LIN {X 0,Y 438.701,Z 233.838,A -85,B 0,C 180,E1 -9266.355,E2 -9266.355} C_VEL
LIN {X 0,Y 435.885,Z 234.19,A -85,B 0,C 180,E1 -9267.602,E2 -9267.602} C_VEL
LIN {X 0,Y 433.569,Z 234.475,A -85,B 0,C 180,E1 -9268.609,E2 -9268.609} C_VEL
LIN {X 0,Y 432.642,Z 234.593,A -85,B 0,C 180,E1 -9269.385,E2 -9269.385} C_VEL
LIN {X 0,Y 432.601,Z 234.596,A -85,B 0,C 180,E1 -9269.648,E2 -9269.648} C_VEL
LIN {X 0,Y 432.582,Z 234.598,A -85,B 0,C 180,E1 -9272.794,E2 -9272.794} C_VEL
LIN {X 0,Y 432.228,Z 234.848,A -85,B 0,C 180,E1 -9275.833,E2 -9275.833} C_VEL
LIN {X 0,Y 432.01,Z 242.324,A -85,B 0,C 180,E1 -9279.362,E2 -9279.362} C_VEL
LIN {X 0,Y 432.001,Z 248.987,A -85,B 0,C 180,E1 -9282.548,E2 -9282.548} C_VEL
LIN {X 0,Y 431.835,Z 256.608,A -85,B 0,C 180,E1 -9286.216,E2 -9286.216} C_VEL
LIN {X 0,Y 431.743,Z 262.883,A -85,B 0,C 180,E1 -9289.241,E2 -9289.241} C_VEL
LIN {X 0,Y 431.628,Z 270.665,A -85,B 0,C 180,E1 -9293.003,E2 -9293.003} C_VEL
LIN {X 0,Y 431.636,Z 272.767,A -85,B 0,C 180,E1 -9294.02,E2 -9294.02} C_VEL
LIN {X 0,Y 433.636,Z 283.694,A -85,B 0,C 180,E1 -9294.477,E2 -9294.477} C_VEL
LIN {X 0,Y 434.113,Z 288.557,A -85,B 0,C 180,E1 -9294.726,E2 -9294.726} C_VEL
LIN {X 0,Y 433.839,Z 297.433,A -85,B 0,C 180,E1 -9295.244,E2 -9295.244} C_VEL
LIN {X 0,Y 433.543,Z 305.193,A -85,B 0,C 180,E1 -9295.814,E2 -9295.814} C_VEL
LIN {X 0,Y 433.148,Z 313.826,A -85,B 0,C 180,E1 -9296.601,E2 -9296.601} C_VEL
LIN {X 0,Y 432.757,Z 322.389,A -85,B 0,C 180,E1 -9297.571,E2 -9297.571} C_VEL
LIN {X 0,Y 432.408,Z 329.809,A -85,B 0,C 180,E1 -9298.637,E2 -9298.637} C_VEL
LIN {X 0,Y 432.074,Z 335.997,A -85,B 0,C 180,E1 -9299.743,E2 -9299.743} C_VEL
LIN {X 0,Y 431.833,Z 341.036,A -85,B 0,C 180,E1 -9300.859,E2 -9300.859} C_VEL
LIN {X 0,Y 431.636,Z 344.371,A -85,B 0,C 180,E1 -9301.763,E2 -9301.763} C_VEL
LIN {X 0,Y 431.505,Z 346.73,A -85,B 0,C 180,E1 -9302.512,E2 -9302.512} C_VEL
LIN {X 0,Y 431.395,Z 349.76,A -85,B 0,C 180,E1 -9303.813,E2 -9303.813} C_VEL
LIN {X 0,Y 431.27,Z 351.381,A -85,B 0,C 180,E1 -9304.776,E2 -9304.776} C_VEL
LIN {X 0,Y 431.202,Z 352.556,A -85,B 0,C 180,E1 -9305.927,E2 -9305.927} C_VEL
LIN {X 0,Y 431.197,Z 352.968,A -85,B 0,C 180,E1 -9307.089,E2 -9307.089} C_VEL
LIN {X 0,Y 431.208,Z 352.366,A -85,B 0,C 180,E1 -9308.526,E2 -9308.526} C_VEL
LIN {X 0,Y 431.279,Z 351.408,A -85,B 0,C 180,E1 -9309.46,E2 -9309.46} C_VEL
LIN {X 0,Y 431.441,Z 349.345,A -85,B 0,C 180,E1 -9310.661,E2 -9310.661} C_VEL
LIN {X 0,Y 431.614,Z 346.292,A -85,B 0,C 180,E1 -9311.883,E2 -9311.883} C_VEL
LIN {X 0,Y 431.882,Z 342.137,A -85,B 0,C 180,E1 -9313.115,E2 -9313.115} C_VEL
LIN {X 0,Y 432.092,Z 337.011,A -85,B 0,C 180,E1 -9314.302,E2 -9314.302} C_VEL
LIN {X 0,Y 432.515,Z 329.674,A -85,B 0,C 180,E1 -9315.64,E2 -9315.64} C_VEL
LIN {X 0,Y 432.986,Z 321.729,A -85,B 0,C 180,E1 -9316.751,E2 -9316.751} C_VEL
LIN {X 0,Y 433.309,Z 314.409,A -85,B 0,C 180,E1 -9317.583,E2 -9317.583} C_VEL
LIN {X 0,Y 433.726,Z 306.857,A -85,B 0,C 180,E1 -9318.285,E2 -9318.285} C_VEL
LIN {X 0,Y 434.003,Z 298.823,A -85,B 0,C 180,E1 -9318.897,E2 -9318.897} C_VEL
LIN {X 0,Y 434.321,Z 289.976,A -85,B 0,C 180,E1 -9319.428,E2 -9319.428} C_VEL
LIN {X 0,Y 434.102,Z 286.131,A -85,B 0,C 180,E1 -9319.639,E2 -9319.639} C_VEL
LIN {X 0,Y 432.039,Z 274.897,A -85,B 0,C 180,E1 -9320.135,E2 -9320.135} C_VEL
LIN {X 0,Y 431.73,Z 273.307,A -85,B 0,C 180,E1 -9320.214,E2 -9320.214} C_VEL
LIN {X 0,Y 431.807,Z 266.369,A -85,B 0,C 180,E1 -9323.554,E2 -9323.554} C_VEL
LIN {X 0,Y 431.884,Z 260.379,A -85,B 0,C 180,E1 -9326.407,E2 -9326.407} C_VEL
LIN {X 0,Y 431.963,Z 255.691,A -85,B 0,C 180,E1 -9328.625,E2 -9328.625} C_VEL
LIN {X 0,Y 432.054,Z 249.71,A -85,B 0,C 180,E1 -9331.449,E2 -9331.449} C_VEL
LIN {X 0,Y 432.147,Z 241.916,A -85,B 0,C 180,E1 -9334.986,E2 -9334.986} C_VEL
LIN {X 0,Y 432.217,Z 234.655,A -85,B 0,C 180,E1 -9338.289,E2 -9338.289} C_VEL
LIN {X 0,Y 432.386,Z 234.628,A -85,B 0,C 180,E1 -9341.029,E2 -9341.029} C_VEL
LIN {X 0,Y 432.433,Z 234.621,A -85,B 0,C 180,E1 -9343.961,E2 -9343.961} C_VEL
LIN {X 0,Y 432.462,Z 234.619,A -85,B 0,C 180,E1 -9347.803,E2 -9347.803} C_VEL
LIN {X 0,Y 432.486,Z 234.615,A -85,B 0,C 180,E1 -9351.59,E2 -9351.59} C_VEL
LIN {X 0,Y 432.583,Z 234.603,A -85,B 0,C 180,E1 -9354.406,E2 -9354.406} C_VEL
LIN {X 0,Y 432.607,Z 234.599,A -85,B 0,C 180,E1 -9358.138,E2 -9358.138} C_VEL
LIN {X 0,Y 432.735,Z 234.583,A -85,B 0,C 180,E1 -9360,E2 -9360} C_VEL
LIN {X 0,Y 432.594,Z 234.601,A -85,B 0,C 180,E1 -9362.794,E2 -9362.794} C_VEL
LIN {X 0,Y 432.588,Z 234.601,A -85,B 0,C 180,E1 -9365.594,E2 -9365.594} C_VEL
LIN {X 0,Y 432.485,Z 234.614,A -85,B 0,C 180,E1 -9368.41,E2 -9368.41} C_VEL
LIN {X 0,Y 432.462,Z 234.618,A -85,B 0,C 180,E1 -9372.196,E2 -9372.196} C_VEL
LIN {X 0,Y 432.433,Z 234.618,A -85,B 0,C 180,E1 -9376.039,E2 -9376.039} C_VEL
LIN {X 0,Y 432.389,Z 234.626,A -85,B 0,C 180,E1 -9379.485,E2 -9379.485} C_VEL
LIN {X 0,Y 432.319,Z 234.635,A -85,B 0,C 180,E1 -9382.964,E2 -9382.964} C_VEL
LIN {X 0,Y 432.352,Z 234.631,A -85,B 0,C 180,E1 -9386.033,E2 -9386.033} C_VEL
LIN {X 0,Y 432.344,Z 234.629,A -85,B 0,C 180,E1 -9389.187,E2 -9389.187} C_VEL
LIN {X 0,Y 432.324,Z 234.634,A -85,B 0,C 180,E1 -9392.443,E2 -9392.443} C_VEL
LIN {X 0,Y 432.344,Z 234.631,A -85,B 0,C 180,E1 -9395.632,E2 -9395.632} C_VEL
LIN {X 0,Y 432.352,Z 234.63,A -85,B 0,C 180,E1 -9399.343,E2 -9399.343} C_VEL
LIN {X 0,Y 432.335,Z 234.632,A -85,B 0,C 180,E1 -9401.797,E2 -9401.797} C_VEL
LIN {X 0,Y 432.335,Z 234.634,A -85,B 0,C 180,E1 -9404.347,E2 -9404.347} C_VEL
LIN {X 0,Y 432.321,Z 234.636,A -85,B 0,C 180,E1 -9407.016,E2 -9407.016} C_VEL
LIN {X 0,Y 432.379,Z 234.679,A -85,B 0,C 180,E1 -9408.391,E2 -9408.391} C_VEL
LIN {X 0,Y 433.342,Z 240.284,A -85,B 0,C 180,E1 -9411.121,E2 -9411.121} C_VEL
LIN {X 0,Y 434.088,Z 244.688,A -85,B 0,C 180,E1 -9413.199,E2 -9413.199} C_VEL
LIN {X 0,Y 434.184,Z 248.536,A -85,B 0,C 180,E1 -9414.926,E2 -9414.926} C_VEL
LIN {X 0,Y 433.596,Z 256.21,A -85,B 0,C 180,E1 -9418.212,E2 -9418.212} C_VEL
LIN {X 0,Y 432.942,Z 265.131,A -85,B 0,C 180,E1 -9421.916,E2 -9421.916} C_VEL
LIN {X 0,Y 432.55,Z 272.79,A -85,B 0,C 180,E1 -9425.011,E2 -9425.011} C_VEL
LIN {X 0,Y 432.083,Z 281.721,A -85,B 0,C 180,E1 -9428.533,E2 -9428.533} C_VEL
LIN {X 0,Y 431.788,Z 289.361,A -85,B 0,C 180,E1 -9431.495,E2 -9431.495} C_VEL
LIN {X 0,Y 431.664,Z 294.798,A -85,B 0,C 180,E1 -9433.555,E2 -9433.555} C_VEL
LIN {X 0,Y 433.565,Z 308.82,A -85,B 0,C 180,E1 -9434.065,E2 -9434.065} C_VEL
LIN {X 0,Y 434.856,Z 320.587,A -85,B 0,C 180,E1 -9434.654,E2 -9434.654} C_VEL
LIN {X 0,Y 434.294,Z 332.166,A -85,B 0,C 180,E1 -9435.354,E2 -9435.354} C_VEL
LIN {X 0,Y 433.643,Z 344.096,A -85,B 0,C 180,E1 -9436.273,E2 -9436.273} C_VEL
LIN {X 0,Y 433.051,Z 355.074,A -85,B 0,C 180,E1 -9437.344,E2 -9437.344} C_VEL
LIN {X 0,Y 432.508,Z 364.833,A -85,B 0,C 180,E1 -9438.518,E2 -9438.518} C_VEL
LIN {X 0,Y 432.017,Z 372.866,A -85,B 0,C 180,E1 -9439.692,E2 -9439.692} C_VEL
LIN {X 0,Y 431.665,Z 380.764,A -85,B 0,C 180,E1 -9441.102,E2 -9441.102} C_VEL
LIN {X 0,Y 431.463,Z 387.072,A -85,B 0,C 180,E1 -9442.513,E2 -9442.513} C_VEL
LIN {X 0,Y 431.296,Z 392.342,A -85,B 0,C 180,E1 -9444.008,E2 -9444.008} C_VEL
LIN {X 0,Y 431.283,Z 395.91,A -85,B 0,C 180,E1 -9445.327,E2 -9445.327} C_VEL
LIN {X 0,Y 431.238,Z 397.871,A -85,B 0,C 180,E1 -9446.262,E2 -9446.262} C_VEL
LIN {X 0,Y 431.318,Z 399.408,A -85,B 0,C 180,E1 -9447.198,E2 -9447.198} C_VEL
LIN {X 0,Y 431.285,Z 400.463,A -85,B 0,C 180,E1 -9448.132,E2 -9448.132} C_VEL
LIN {X 0,Y 431.292,Z 401.104,A -85,B 0,C 180,E1 -9449.066,E2 -9449.066} C_VEL
LIN {X 0,Y 431.283,Z 401.338,A -85,B 0,C 180,E1 -9450,E2 -9450} C_VEL
LIN {X 0,Y 431.262,Z 401.157,A -85,B 0,C 180,E1 -9450.934,E2 -9450.934} C_VEL
LIN {X 0,Y 431.274,Z 400.52,A -85,B 0,C 180,E1 -9451.868,E2 -9451.868} C_VEL
LIN {X 0,Y 431.318,Z 399.475,A -85,B 0,C 180,E1 -9452.802,E2 -9452.802} C_VEL
LIN {X 0,Y 431.23,Z 398.014,A -85,B 0,C 180,E1 -9453.738,E2 -9453.738} C_VEL
LIN {X 0,Y 431.322,Z 394.966,A -85,B 0,C 180,E1 -9455.142,E2 -9455.142} C_VEL
LIN {X 0,Y 431.376,Z 390.847,A -85,B 0,C 180,E1 -9456.549,E2 -9456.549} C_VEL
LIN {X 0,Y 431.582,Z 384.552,A -85,B 0,C 180,E1 -9458.192,E2 -9458.192} C_VEL
LIN {X 0,Y 431.856,Z 377.702,A -85,B 0,C 180,E1 -9459.602,E2 -9459.602} C_VEL
LIN {X 0,Y 432.322,Z 369.259,A -85,B 0,C 180,E1 -9461.012,E2 -9461.012} C_VEL
LIN {X 0,Y 432.9,Z 360.702,A -85,B 0,C 180,E1 -9462.184,E2 -9462.184} C_VEL
LIN {X 0,Y 433.391,Z 351.217,A -85,B 0,C 180,E1 -9463.267,E2 -9463.267} C_VEL
LIN {X 0,Y 434.171,Z 340.199,A -85,B 0,C 180,E1 -9464.292,E2 -9464.292} C_VEL
LIN {X 0,Y 435.046,Z 327.759,A -85,B 0,C 180,E1 -9465.219,E2 -9465.219} C_VEL
LIN {X 0,Y 435.258,Z 320.109,A -85,B 0,C 180,E1 -9465.692,E2 -9465.692} C_VEL
LIN {X 0,Y 434.242,Z 307.284,A -85,B 0,C 180,E1 -9466.395,E2 -9466.395} C_VEL
LIN {X 0,Y 432.159,Z 294.828,A -85,B 0,C 180,E1 -9466.968,E2 -9466.968} C_VEL
LIN {X 0,Y 431.597,Z 291.722,A -85,B 0,C 180,E1 -9467.105,E2 -9467.105} C_VEL
LIN {X 0,Y 431.878,Z 282.941,A -85,B 0,C 180,E1 -9470.48,E2 -9470.48} C_VEL
LIN {X 0,Y 432.213,Z 275.478,A -85,B 0,C 180,E1 -9473.477,E2 -9473.477} C_VEL
LIN {X 0,Y 432.667,Z 267.899,A -85,B 0,C 180,E1 -9476.697,E2 -9476.697} C_VEL
LIN {X 0,Y 433.186,Z 261.43,A -85,B 0,C 180,E1 -9479.659,E2 -9479.659} C_VEL
LIN {X 0,Y 433.901,Z 255.542,A -85,B 0,C 180,E1 -9482.621,E2 -9482.621} C_VEL
LIN {X 0,Y 434.361,Z 252.169,A -85,B 0,C 180,E1 -9484.493,E2 -9484.493} C_VEL
LIN {X 0,Y 434.538,Z 248.602,A -85,B 0,C 180,E1 -9486.757,E2 -9486.757} C_VEL
LIN {X 0,Y 434.258,Z 245.52,A -85,B 0,C 180,E1 -9489.137,E2 -9489.137} C_VEL
LIN {X 0,Y 433.805,Z 242.819,A -85,B 0,C 180,E1 -9491.82,E2 -9491.82} C_VEL
LIN {X 0,Y 433.477,Z 240.907,A -85,B 0,C 180,E1 -9494.49,E2 -9494.49} C_VEL
LIN {X 0,Y 433.227,Z 239.772,A -85,B 0,C 180,E1 -9497.051,E2 -9497.051} C_VEL
LIN {X 0,Y 433.123,Z 239.257,A -85,B 0,C 180,E1 -9499.698,E2 -9499.698} C_VEL
LIN {X 0,Y 433.098,Z 239.446,A -85,B 0,C 180,E1 -9503.101,E2 -9503.101} C_VEL
LIN {X 0,Y 433.01,Z 240.207,A -85,B 0,C 180,E1 -9505.87,E2 -9505.87} C_VEL
LIN {X 0,Y 432.715,Z 241.447,A -85,B 0,C 180,E1 -9508.686,E2 -9508.686} C_VEL
LIN {X 0,Y 432.439,Z 243.225,A -85,B 0,C 180,E1 -9511.881,E2 -9511.881} C_VEL
LIN {X 0,Y 432.306,Z 244.571,A -85,B 0,C 180,E1 -9513.964,E2 -9513.964} C_VEL
LIN {X 0,Y 432.089,Z 246.753,A -85,B 0,C 180,E1 -9517.023,E2 -9517.023} C_VEL
LIN {X 0,Y 431.942,Z 249.63,A -85,B 0,C 180,E1 -9520.684,E2 -9520.684} C_VEL
LIN {X 0,Y 431.881,Z 252.494,A -85,B 0,C 180,E1 -9524.061,E2 -9524.061} C_VEL
LIN {X 0,Y 435.436,Z 264.773,A -85,B 0,C 180,E1 -9524.753,E2 -9524.753} C_VEL
LIN {X 0,Y 436.678,Z 271.049,A -85,B 0,C 180,E1 -9525.137,E2 -9525.137} C_VEL
LIN {X 0,Y 435.976,Z 283.695,A -85,B 0,C 180,E1 -9525.887,E2 -9525.887} C_VEL
LIN {X 0,Y 435.237,Z 295.639,A -85,B 0,C 180,E1 -9526.816,E2 -9526.816} C_VEL
LIN {X 0,Y 434.487,Z 306.414,A -85,B 0,C 180,E1 -9527.861,E2 -9527.861} C_VEL
LIN {X 0,Y 433.871,Z 316.104,A -85,B 0,C 180,E1 -9529.028,E2 -9529.028} C_VEL
LIN {X 0,Y 433.179,Z 325.539,A -85,B 0,C 180,E1 -9530.427,E2 -9530.427} C_VEL
LIN {X 0,Y 432.616,Z 333.133,A -85,B 0,C 180,E1 -9531.828,E2 -9531.828} C_VEL
LIN {X 0,Y 432.043,Z 340.11,A -85,B 0,C 180,E1 -9533.462,E2 -9533.462} C_VEL
LIN {X 0,Y 431.926,Z 344.73,A -85,B 0,C 180,E1 -9534.866,E2 -9534.866} C_VEL
LIN {X 0,Y 431.807,Z 348.254,A -85,B 0,C 180,E1 -9536.267,E2 -9536.267} C_VEL
LIN {X 0,Y 431.621,Z 350.072,A -85,B 0,C 180,E1 -9537.2,E2 -9537.2} C_VEL
LIN {X 0,Y 431.429,Z 351.421,A -85,B 0,C 180,E1 -9538.133,E2 -9538.133} C_VEL
LIN {X 0,Y 431.292,Z 352.894,A -85,B 0,C 180,E1 -9540,E2 -9540} C_VEL
LIN {X 0,Y 431.316,Z 353.025,A -85,B 0,C 180,E1 -9540.934,E2 -9540.934} C_VEL
LIN {X 0,Y 431.395,Z 352.011,A -85,B 0,C 180,E1 -9542.802,E2 -9542.802} C_VEL
LIN {X 0,Y 431.442,Z 350.912,A -85,B 0,C 180,E1 -9543.736,E2 -9543.736} C_VEL
LIN {X 0,Y 431.389,Z 349.378,A -85,B 0,C 180,E1 -9544.672,E2 -9544.672} C_VEL
LIN {X 0,Y 431.596,Z 346.24,A -85,B 0,C 180,E1 -9546.076,E2 -9546.076} C_VEL
LIN {X 0,Y 431.705,Z 342.027,A -85,B 0,C 180,E1 -9547.483,E2 -9547.483} C_VEL
LIN {X 0,Y 432.065,Z 335.576,A -85,B 0,C 180,E1 -9549.125,E2 -9549.125} C_VEL
LIN {X 0,Y 432.393,Z 328.569,A -85,B 0,C 180,E1 -9550.536,E2 -9550.536} C_VEL
LIN {X 0,Y 432.936,Z 319.801,A -85,B 0,C 180,E1 -9551.945,E2 -9551.945} C_VEL
LIN {X 0,Y 433.438,Z 309.685,A -85,B 0,C 180,E1 -9553.261,E2 -9553.261} C_VEL
LIN {X 0,Y 433.962,Z 299.835,A -85,B 0,C 180,E1 -9554.299,E2 -9554.299} C_VEL
LIN {X 0,Y 434.644,Z 288.818,A -85,B 0,C 180,E1 -9555.234,E2 -9555.234} C_VEL
LIN {X 0,Y 435.221,Z 276.122,A -85,B 0,C 180,E1 -9556.09,E2 -9556.09} C_VEL
LIN {X 0,Y 435.287,Z 267.404,A -85,B 0,C 180,E1 -9556.556,E2 -9556.556} C_VEL
LIN {X 0,Y 432.494,Z 254.275,A -85,B 0,C 180,E1 -9557.189,E2 -9557.189} C_VEL
LIN {X 0,Y 431.416,Z 249.122,A -85,B 0,C 180,E1 -9557.406,E2 -9557.406} C_VEL
LIN {X 0,Y 431.412,Z 246.253,A -85,B 0,C 180,E1 -9560.005,E2 -9560.005} C_VEL
LIN {X 0,Y 431.424,Z 242.986,A -85,B 0,C 180,E1 -9563.015,E2 -9563.015} C_VEL
LIN {X 0,Y 431.602,Z 239.361,A -85,B 0,C 180,E1 -9566.414,E2 -9566.414} C_VEL
LIN {X 0,Y 431.597,Z 236.411,A -85,B 0,C 180,E1 -9569.243,E2 -9569.243} C_VEL
LIN {X 0,Y 431.615,Z 235.278,A -85,B 0,C 180,E1 -9570.344,E2 -9570.344} C_VEL
LIN {X 0,Y 431.687,Z 234.716,A -85,B 0,C 180,E1 -9571.398,E2 -9571.398} C_VEL
LIN {X 0,Y 432.087,Z 234.664,A -85,B 0,C 180,E1 -9574.701,E2 -9574.701} C_VEL
LIN {X 0,Y 432.29,Z 234.637,A -85,B 0,C 180,E1 -9577.191,E2 -9577.191} C_VEL
LIN {X 0,Y 432.336,Z 234.631,A -85,B 0,C 180,E1 -9580.179,E2 -9580.179} C_VEL
LIN {X 0,Y 432.318,Z 234.634,A -85,B 0,C 180,E1 -9583.061,E2 -9583.061} C_VEL
LIN {X 0,Y 432.336,Z 234.631,A -85,B 0,C 180,E1 -9585.665,E2 -9585.665} C_VEL
LIN {X 0,Y 432.315,Z 234.632,A -85,B 0,C 180,E1 -9588.401,E2 -9588.401} C_VEL
LIN {X 0,Y 432.324,Z 234.63,A -85,B 0,C 180,E1 -9591.848,E2 -9591.848} C_VEL
LIN {X 0,Y 432.328,Z 234.63,A -85,B 0,C 180,E1 -9595.321,E2 -9595.321} C_VEL
LIN {X 0,Y 432.323,Z 234.635,A -85,B 0,C 180,E1 -9598.654,E2 -9598.654} C_VEL
LIN {X 0,Y 432.351,Z 234.629,A -85,B 0,C 180,E1 -9601.874,E2 -9601.874} C_VEL
LIN {X 0,Y 432.383,Z 234.625,A -85,B 0,C 180,E1 -9605.538,E2 -9605.538} C_VEL
LIN {X 0,Y 432.354,Z 234.629,A -85,B 0,C 180,E1 -9609.046,E2 -9609.046} C_VEL
LIN {X 0,Y 432.365,Z 234.628,A -85,B 0,C 180,E1 -9612.01,E2 -9612.01} C_VEL
LIN {X 0,Y 432.398,Z 234.624,A -85,B 0,C 180,E1 -9614.926,E2 -9614.926} C_VEL
LIN {X 0,Y 432.463,Z 234.615,A -85,B 0,C 180,E1 -9617.803,E2 -9617.803} C_VEL
LIN {X 0,Y 432.465,Z 234.614,A -85,B 0,C 180,E1 -9621.59,E2 -9621.59} C_VEL
LIN {X 0,Y 432.55,Z 234.604,A -85,B 0,C 180,E1 -9624.405,E2 -9624.405} C_VEL
LIN {X 0,Y 432.598,Z 234.598,A -85,B 0,C 180,E1 -9628.138,E2 -9628.138} C_VEL
LIN {X 0,Y 432.601,Z 234.596,A -85,B 0,C 180,E1 -9629.648,E2 -9629.648} C_VEL
LIN {X 0,Y 432.018,Z 234.672,A -85,B 0,C 180,E1 -9630.425,E2 -9630.425} C_VEL
LIN {X 0,Y 429.144,Z 235.031,A -85,B 0,C 180,E1 -9631.686,E2 -9631.686} C_VEL
LIN {X 0,Y 426.601,Z 235.344,A -85,B 0,C 180,E1 -9632.704,E2 -9632.704} C_VEL
LIN {X 0,Y 425.43,Z 235.495,A -85,B 0,C 180,E1 -9633.491,E2 -9633.491} C_VEL
LIN {X 0,Y 425.297,Z 235.508,A -85,B 0,C 180,E1 -9633.759,E2 -9633.759} C_VEL
LIN {X 0,Y 425.162,Z 235.561,A -85,B 0,C 180,E1 -9635.692,E2 -9635.692} C_VEL
LIN {X 0,Y 424.964,Z 242.559,A -85,B 0,C 180,E1 -9639.039,E2 -9639.039} C_VEL
LIN {X 0,Y 424.959,Z 250.045,A -85,B 0,C 180,E1 -9642.643,E2 -9642.643} C_VEL
LIN {X 0,Y 424.775,Z 257.688,A -85,B 0,C 180,E1 -9646.336,E2 -9646.336} C_VEL
LIN {X 0,Y 424.66,Z 263.961,A -85,B 0,C 180,E1 -9649.38,E2 -9649.38} C_VEL
LIN {X 0,Y 424.577,Z 271.188,A -85,B 0,C 180,E1 -9652.892,E2 -9652.892} C_VEL
LIN {X 0,Y 424.581,Z 273.154,A -85,B 0,C 180,E1 -9653.828,E2 -9653.828} C_VEL
LIN {X 0,Y 426.406,Z 283.093,A -85,B 0,C 180,E1 -9654.236,E2 -9654.236} C_VEL
LIN {X 0,Y 427.21,Z 288.257,A -85,B 0,C 180,E1 -9654.503,E2 -9654.503} C_VEL
LIN {X 0,Y 426.932,Z 297.133,A -85,B 0,C 180,E1 -9655.02,E2 -9655.02} C_VEL
LIN {X 0,Y 426.602,Z 305.304,A -85,B 0,C 180,E1 -9655.623,E2 -9655.623} C_VEL
LIN {X 0,Y 426.257,Z 312.787,A -85,B 0,C 180,E1 -9656.302,E2 -9656.302} C_VEL
LIN {X 0,Y 425.877,Z 321.025,A -85,B 0,C 180,E1 -9657.22,E2 -9657.22} C_VEL
LIN {X 0,Y 425.459,Z 329.228,A -85,B 0,C 180,E1 -9658.354,E2 -9658.354} C_VEL
LIN {X 0,Y 425.077,Z 335.705,A -85,B 0,C 180,E1 -9659.498,E2 -9659.498} C_VEL
LIN {X 0,Y 424.8,Z 340.932,A -85,B 0,C 180,E1 -9660.649,E2 -9660.649} C_VEL
LIN {X 0,Y 424.617,Z 343.917,A -85,B 0,C 180,E1 -9661.424,E2 -9661.424} C_VEL
LIN {X 0,Y 424.453,Z 346.93,A -85,B 0,C 180,E1 -9662.387,E2 -9662.387} C_VEL
LIN {X 0,Y 424.259,Z 350.658,A -85,B 0,C 180,E1 -9664.078,E2 -9664.078} C_VEL
LIN {X 0,Y 424.134,Z 352.758,A -85,B 0,C 180,E1 -9665.713,E2 -9665.713} C_VEL
LIN {X 0,Y 424.095,Z 353.316,A -85,B 0,C 180,E1 -9667.302,E2 -9667.302} C_VEL
LIN {X 0,Y 424.173,Z 352.308,A -85,B 0,C 180,E1 -9669.021,E2 -9669.021} C_VEL
LIN {X 0,Y 424.312,Z 350.407,A -85,B 0,C 180,E1 -9670.366,E2 -9670.366} C_VEL
LIN {X 0,Y 424.542,Z 347.073,A -85,B 0,C 180,E1 -9671.845,E2 -9671.845} C_VEL
LIN {X 0,Y 424.847,Z 342.276,A -85,B 0,C 180,E1 -9673.292,E2 -9673.292} C_VEL
LIN {X 0,Y 425.061,Z 337.824,A -85,B 0,C 180,E1 -9674.344,E2 -9674.344} C_VEL
LIN {X 0,Y 425.336,Z 333.04,A -85,B 0,C 180,E1 -9675.276,E2 -9675.276} C_VEL
LIN {X 0,Y 425.709,Z 326.72,A -85,B 0,C 180,E1 -9676.293,E2 -9676.293} C_VEL
LIN {X 0,Y 426.131,Z 319.718,A -85,B 0,C 180,E1 -9677.216,E2 -9677.216} C_VEL
LIN {X 0,Y 426.669,Z 310.622,A -85,B 0,C 180,E1 -9678.189,E2 -9678.189} C_VEL
LIN {X 0,Y 427.024,Z 301.67,A -85,B 0,C 180,E1 -9678.938,E2 -9678.938} C_VEL
LIN {X 0,Y 427.399,Z 291.666,A -85,B 0,C 180,E1 -9679.575,E2 -9679.575} C_VEL
LIN {X 0,Y 427.164,Z 286.681,A -85,B 0,C 180,E1 -9679.855,E2 -9679.855} C_VEL
LIN {X 0,Y 424.973,Z 275.153,A -85,B 0,C 180,E1 -9680.377,E2 -9680.377} C_VEL
LIN {X 0,Y 424.696,Z 273.649,A -85,B 0,C 180,E1 -9680.461,E2 -9680.461} C_VEL
LIN {X 0,Y 424.769,Z 267.47,A -85,B 0,C 180,E1 -9683.442,E2 -9683.442} C_VEL
LIN {X 0,Y 424.848,Z 261.382,A -85,B 0,C 180,E1 -9686.361,E2 -9686.361} C_VEL
LIN {X 0,Y 424.967,Z 254.302,A -85,B 0,C 180,E1 -9689.79,E2 -9689.79} C_VEL
LIN {X 0,Y 425.015,Z 248.557,A -85,B 0,C 180,E1 -9692.419,E2 -9692.419} C_VEL
LIN {X 0,Y 425.155,Z 240.485,A -85,B 0,C 180,E1 -9696.109,E2 -9696.109} C_VEL
LIN {X 0,Y 425.181,Z 235.53,A -85,B 0,C 180,E1 -9698.427,E2 -9698.427} C_VEL
LIN {X 0,Y 425.361,Z 235.503,A -85,B 0,C 180,E1 -9700.704,E2 -9700.704} C_VEL
LIN {X 0,Y 425.391,Z 235.499,A -85,B 0,C 180,E1 -9703.688,E2 -9703.688} C_VEL
LIN {X 0,Y 425.415,Z 235.496,A -85,B 0,C 180,E1 -9707.598,E2 -9707.598} C_VEL
LIN {X 0,Y 425.44,Z 235.492,A -85,B 0,C 180,E1 -9711.45,E2 -9711.45} C_VEL
LIN {X 0,Y 425.537,Z 235.481,A -85,B 0,C 180,E1 -9714.313,E2 -9714.313} C_VEL
LIN {X 0,Y 425.576,Z 235.475,A -85,B 0,C 180,E1 -9718.107,E2 -9718.107} C_VEL
LIN {X 0,Y 425.705,Z 235.459,A -85,B 0,C 180,E1 -9720,E2 -9720} C_VEL
LIN {X 0,Y 425.548,Z 235.479,A -85,B 0,C 180,E1 -9722.84,E2 -9722.84} C_VEL
LIN {X 0,Y 425.543,Z 235.479,A -85,B 0,C 180,E1 -9725.687,E2 -9725.687} C_VEL
LIN {X 0,Y 425.439,Z 235.491,A -85,B 0,C 180,E1 -9728.55,E2 -9728.55} C_VEL
LIN {X 0,Y 425.415,Z 235.495,A -85,B 0,C 180,E1 -9732.402,E2 -9732.402} C_VEL
LIN {X 0,Y 425.39,Z 235.495,A -85,B 0,C 180,E1 -9736.312,E2 -9736.312} C_VEL
LIN {X 0,Y 425.33,Z 235.505,A -85,B 0,C 180,E1 -9739.635,E2 -9739.635} C_VEL
LIN {X 0,Y 425.29,Z 235.51,A -85,B 0,C 180,E1 -9742.339,E2 -9742.339} C_VEL
LIN {X 0,Y 425.322,Z 235.505,A -85,B 0,C 180,E1 -9744.657,E2 -9744.657} C_VEL
LIN {X 0,Y 425.347,Z 235.504,A -85,B 0,C 180,E1 -9747.558,E2 -9747.558} C_VEL
LIN {X 0,Y 425.289,Z 235.511,A -85,B 0,C 180,E1 -9750.816,E2 -9750.816} C_VEL
LIN {X 0,Y 425.311,Z 235.507,A -85,B 0,C 180,E1 -9754.288,E2 -9754.288} C_VEL
LIN {X 0,Y 425.281,Z 235.51,A -85,B 0,C 180,E1 -9757.694,E2 -9757.694} C_VEL
LIN {X 0,Y 425.283,Z 235.512,A -85,B 0,C 180,E1 -9760.521,E2 -9760.521} C_VEL
LIN {X 0,Y 425.259,Z 235.514,A -85,B 0,C 180,E1 -9763.351,E2 -9763.351} C_VEL
LIN {X 0,Y 425.259,Z 235.516,A -85,B 0,C 180,E1 -9766.649,E2 -9766.649} C_VEL
LIN {X 0,Y 425.379,Z 235.717,A -85,B 0,C 180,E1 -9768.231,E2 -9768.231} C_VEL
LIN {X 0,Y 426.41,Z 241.753,A -85,B 0,C 180,E1 -9771.222,E2 -9771.222} C_VEL
LIN {X 0,Y 427.176,Z 247.015,A -85,B 0,C 180,E1 -9773.723,E2 -9773.723} C_VEL
LIN {X 0,Y 426.988,Z 252.044,A -85,B 0,C 180,E1 -9775.97,E2 -9775.97} C_VEL
LIN {X 0,Y 426.39,Z 259.043,A -85,B 0,C 180,E1 -9778.992,E2 -9778.992} C_VEL
LIN {X 0,Y 425.801,Z 267.331,A -85,B 0,C 180,E1 -9782.474,E2 -9782.474} C_VEL
LIN {X 0,Y 425.374,Z 274.961,A -85,B 0,C 180,E1 -9785.604,E2 -9785.604} C_VEL
LIN {X 0,Y 425,Z 282.574,A -85,B 0,C 180,E1 -9788.666,E2 -9788.666} C_VEL
LIN {X 0,Y 424.693,Z 290.197,A -85,B 0,C 180,E1 -9791.674,E2 -9791.674} C_VEL
LIN {X 0,Y 424.581,Z 294.613,A -85,B 0,C 180,E1 -9793.33,E2 -9793.33} C_VEL
LIN {X 0,Y 426.498,Z 308.655,A -85,B 0,C 180,E1 -9793.855,E2 -9793.855} C_VEL
LIN {X 0,Y 427.892,Z 321.46,A -85,B 0,C 180,E1 -9794.52,E2 -9794.52} C_VEL
LIN {X 0,Y 427.167,Z 334.441,A -85,B 0,C 180,E1 -9795.347,E2 -9795.347} C_VEL
LIN {X 0,Y 426.52,Z 345.913,A -85,B 0,C 180,E1 -9796.299,E2 -9796.299} C_VEL
LIN {X 0,Y 425.868,Z 357.402,A -85,B 0,C 180,E1 -9797.491,E2 -9797.491} C_VEL
LIN {X 0,Y 425.303,Z 367.474,A -85,B 0,C 180,E1 -9798.804,E2 -9798.804} C_VEL
LIN {X 0,Y 424.811,Z 376.357,A -85,B 0,C 180,E1 -9800.237,E2 -9800.237} C_VEL
LIN {X 0,Y 424.507,Z 383.482,A -85,B 0,C 180,E1 -9801.671,E2 -9801.671} C_VEL
LIN {X 0,Y 424.299,Z 389.976,A -85,B 0,C 180,E1 -9803.342,E2 -9803.342} C_VEL
LIN {X 0,Y 424.251,Z 394.233,A -85,B 0,C 180,E1 -9804.773,E2 -9804.773} C_VEL
LIN {X 0,Y 424.146,Z 397.378,A -85,B 0,C 180,E1 -9806.2,E2 -9806.2} C_VEL
LIN {X 0,Y 424.246,Z 398.935,A -85,B 0,C 180,E1 -9807.151,E2 -9807.151} C_VEL
LIN {X 0,Y 424.207,Z 400.018,A -85,B 0,C 180,E1 -9808.101,E2 -9808.101} C_VEL
LIN {X 0,Y 424.204,Z 400.671,A -85,B 0,C 180,E1 -9809.051,E2 -9809.051} C_VEL
LIN {X 0,Y 424.208,Z 400.92,A -85,B 0,C 180,E1 -9810,E2 -9810} C_VEL
LIN {X 0,Y 424.177,Z 400.757,A -85,B 0,C 180,E1 -9810.95,E2 -9810.95} C_VEL
LIN {X 0,Y 424.197,Z 400.141,A -85,B 0,C 180,E1 -9811.899,E2 -9811.899} C_VEL
LIN {X 0,Y 424.227,Z 399.106,A -85,B 0,C 180,E1 -9812.849,E2 -9812.849} C_VEL
LIN {X 0,Y 424.138,Z 397.651,A -85,B 0,C 180,E1 -9813.801,E2 -9813.801} C_VEL
LIN {X 0,Y 424.23,Z 394.627,A -85,B 0,C 180,E1 -9815.228,E2 -9815.228} C_VEL
LIN {X 0,Y 424.299,Z 390.537,A -85,B 0,C 180,E1 -9816.658,E2 -9816.658} C_VEL
LIN {X 0,Y 424.505,Z 384.295,A -85,B 0,C 180,E1 -9818.33,E2 -9818.33} C_VEL
LIN {X 0,Y 424.902,Z 376.208,A -85,B 0,C 180,E1 -9820.002,E2 -9820.002} C_VEL
LIN {X 0,Y 425.492,Z 367.534,A -85,B 0,C 180,E1 -9821.432,E2 -9821.432} C_VEL
LIN {X 0,Y 426.123,Z 356.74,A -85,B 0,C 180,E1 -9822.865,E2 -9822.865} C_VEL
LIN {X 0,Y 426.872,Z 345.863,A -85,B 0,C 180,E1 -9824.03,E2 -9824.03} C_VEL
LIN {X 0,Y 427.835,Z 333.115,A -85,B 0,C 180,E1 -9825.116,E2 -9825.116} C_VEL
LIN {X 0,Y 428.57,Z 322.743,A -85,B 0,C 180,E1 -9825.821,E2 -9825.821} C_VEL
LIN {X 0,Y 427.706,Z 310.377,A -85,B 0,C 180,E1 -9826.561,E2 -9826.561} C_VEL
LIN {X 0,Y 426.003,Z 298.748,A -85,B 0,C 180,E1 -9827.15,E2 -9827.15} C_VEL
LIN {X 0,Y 424.546,Z 291.222,A -85,B 0,C 180,E1 -9827.492,E2 -9827.492} C_VEL
LIN {X 0,Y 424.874,Z 282.753,A -85,B 0,C 180,E1 -9830.833,E2 -9830.833} C_VEL
LIN {X 0,Y 425.202,Z 275.358,A -85,B 0,C 180,E1 -9833.888,E2 -9833.888} C_VEL
LIN {X 0,Y 425.676,Z 268.411,A -85,B 0,C 180,E1 -9836.931,E2 -9836.931} C_VEL
LIN {X 0,Y 426.275,Z 261.541,A -85,B 0,C 180,E1 -9840.189,E2 -9840.189} C_VEL
LIN {X 0,Y 426.99,Z 256.312,A -85,B 0,C 180,E1 -9842.92,E2 -9842.92} C_VEL
LIN {X 0,Y 427.468,Z 252.528,A -85,B 0,C 180,E1 -9845.131,E2 -9845.131} C_VEL
LIN {X 0,Y 427.56,Z 249.108,A -85,B 0,C 180,E1 -9847.459,E2 -9847.459} C_VEL
LIN {X 0,Y 427.177,Z 246.189,A -85,B 0,C 180,E1 -9849.914,E2 -9849.914} C_VEL
LIN {X 0,Y 426.761,Z 243.856,A -85,B 0,C 180,E1 -9852.47,E2 -9852.47} C_VEL
LIN {X 0,Y 426.461,Z 242.122,A -85,B 0,C 180,E1 -9855.124,E2 -9855.124} C_VEL
LIN {X 0,Y 426.262,Z 241.066,A -85,B 0,C 180,E1 -9857.897,E2 -9857.897} C_VEL
LIN {X 0,Y 426.168,Z 240.691,A -85,B 0,C 180,E1 -9861.195,E2 -9861.195} C_VEL
LIN {X 0,Y 426.121,Z 241.009,A -85,B 0,C 180,E1 -9863.917,E2 -9863.917} C_VEL
LIN {X 0,Y 426.032,Z 241.551,A -85,B 0,C 180,E1 -9865.883,E2 -9865.883} C_VEL
LIN {X 0,Y 425.693,Z 242.954,A -85,B 0,C 180,E1 -9869.216,E2 -9869.216} C_VEL
LIN {X 0,Y 425.398,Z 244.746,A -85,B 0,C 180,E1 -9872.446,E2 -9872.446} C_VEL
LIN {X 0,Y 425.205,Z 246.789,A -85,B 0,C 180,E1 -9875.593,E2 -9875.593} C_VEL
LIN {X 0,Y 424.957,Z 249.036,A -85,B 0,C 180,E1 -9878.664,E2 -9878.664} C_VEL
LIN {X 0,Y 424.862,Z 251.418,A -85,B 0,C 180,E1 -9881.682,E2 -9881.682} C_VEL
LIN {X 0,Y 424.864,Z 253.285,A -85,B 0,C 180,E1 -9883.683,E2 -9883.683} C_VEL
LIN {X 0,Y 428.378,Z 264.542,A -85,B 0,C 180,E1 -9884.351,E2 -9884.351} C_VEL
LIN {X 0,Y 430.013,Z 272.165,A -85,B 0,C 180,E1 -9884.841,E2 -9884.841} C_VEL
LIN {X 0,Y 429.346,Z 283.394,A -85,B 0,C 180,E1 -9885.521,E2 -9885.521} C_VEL
LIN {X 0,Y 428.544,Z 295.698,A -85,B 0,C 180,E1 -9886.485,E2 -9886.485} C_VEL
LIN {X 0,Y 427.73,Z 306.504,A -85,B 0,C 180,E1 -9887.546,E2 -9887.546} C_VEL
LIN {X 0,Y 427.099,Z 315.381,A -85,B 0,C 180,E1 -9888.611,E2 -9888.611} C_VEL
LIN {X 0,Y 426.351,Z 324.995,A -85,B 0,C 180,E1 -9890.033,E2 -9890.033} C_VEL
LIN {X 0,Y 425.702,Z 332.781,A -85,B 0,C 180,E1 -9891.455,E2 -9891.455} C_VEL
LIN {X 0,Y 425.198,Z 339.247,A -85,B 0,C 180,E1 -9892.934,E2 -9892.934} C_VEL
LIN {X 0,Y 425.018,Z 343.98,A -85,B 0,C 180,E1 -9894.306,E2 -9894.306} C_VEL
LIN {X 0,Y 424.798,Z 347.809,A -85,B 0,C 180,E1 -9895.731,E2 -9895.731} C_VEL
LIN {X 0,Y 424.578,Z 350.616,A -85,B 0,C 180,E1 -9897.154,E2 -9897.154} C_VEL
LIN {X 0,Y 424.265,Z 352.835,A -85,B 0,C 180,E1 -9899.051,E2 -9899.051} C_VEL
LIN {X 0,Y 424.233,Z 353.346,A -85,B 0,C 180,E1 -9900,E2 -9900} C_VEL
LIN {X 0,Y 424.228,Z 353.43,A -85,B 0,C 180,E1 -9900.949,E2 -9900.949} C_VEL
LIN {X 0,Y 424.326,Z 352.356,A -85,B 0,C 180,E1 -9902.848,E2 -9902.848} C_VEL
LIN {X 0,Y 424.348,Z 351.227,A -85,B 0,C 180,E1 -9903.799,E2 -9903.799} C_VEL
LIN {X 0,Y 424.394,Z 348.696,A -85,B 0,C 180,E1 -9905.226,E2 -9905.226} C_VEL
LIN {X 0,Y 424.549,Z 344.55,A -85,B 0,C 180,E1 -9906.851,E2 -9906.851} C_VEL
LIN {X 0,Y 424.745,Z 340.484,A -85,B 0,C 180,E1 -9908.085,E2 -9908.085} C_VEL
LIN {X 0,Y 425.124,Z 333.413,A -85,B 0,C 180,E1 -9909.756,E2 -9909.756} C_VEL
LIN {X 0,Y 425.546,Z 325.769,A -85,B 0,C 180,E1 -9911.19,E2 -9911.19} C_VEL
LIN {X 0,Y 426.084,Z 317.986,A -85,B 0,C 180,E1 -9912.382,E2 -9912.382} C_VEL
LIN {X 0,Y 426.577,Z 307.694,A -85,B 0,C 180,E1 -9913.672,E2 -9913.672} C_VEL
LIN {X 0,Y 427.205,Z 296.808,A -85,B 0,C 180,E1 -9914.773,E2 -9914.773} C_VEL
LIN {X 0,Y 427.917,Z 284.969,A -85,B 0,C 180,E1 -9915.723,E2 -9915.723} C_VEL
LIN {X 0,Y 428.449,Z 272.002,A -85,B 0,C 180,E1 -9916.533,E2 -9916.533} C_VEL
LIN {X 0,Y 428.268,Z 268.033,A -85,B 0,C 180,E1 -9916.745,E2 -9916.745} C_VEL
LIN {X 0,Y 425.408,Z 254.565,A -85,B 0,C 180,E1 -9917.408,E2 -9917.408} C_VEL
LIN {X 0,Y 424.335,Z 249.464,A -85,B 0,C 180,E1 -9917.625,E2 -9917.625} C_VEL
LIN {X 0,Y 424.352,Z 246.471,A -85,B 0,C 180,E1 -9920.353,E2 -9920.353} C_VEL
LIN {X 0,Y 424.349,Z 243.177,A -85,B 0,C 180,E1 -9923.421,E2 -9923.421} C_VEL
LIN {X 0,Y 424.541,Z 239.777,A -85,B 0,C 180,E1 -9926.627,E2 -9926.627} C_VEL
LIN {X 0,Y 424.528,Z 236.518,A -85,B 0,C 180,E1 -9929.779,E2 -9929.779} C_VEL
LIN {X 0,Y 424.563,Z 235.603,A -85,B 0,C 180,E1 -9930.875,E2 -9930.875} C_VEL
LIN {X 0,Y 425.001,Z 235.545,A -85,B 0,C 180,E1 -9934.226,E2 -9934.226} C_VEL
LIN {X 0,Y 425.202,Z 235.52,A -85,B 0,C 180,E1 -9936.515,E2 -9936.515} C_VEL
LIN {X 0,Y 425.277,Z 235.511,A -85,B 0,C 180,E1 -9939.039,E2 -9939.039} C_VEL
LIN {X 0,Y 425.286,Z 235.509,A -85,B 0,C 180,E1 -9941.957,E2 -9941.957} C_VEL
LIN {X 0,Y 425.288,Z 235.512,A -85,B 0,C 180,E1 -9945.283,E2 -9945.283} C_VEL
LIN {X 0,Y 425.254,Z 235.513,A -85,B 0,C 180,E1 -9948.618,E2 -9948.618} C_VEL
LIN {X 0,Y 425.278,Z 235.512,A -85,B 0,C 180,E1 -9951.099,E2 -9951.099} C_VEL
LIN {X 0,Y 425.295,Z 235.511,A -85,B 0,C 180,E1 -9954.663,E2 -9954.663} C_VEL
LIN {X 0,Y 425.266,Z 235.511,A -85,B 0,C 180,E1 -9958.073,E2 -9958.073} C_VEL
LIN {X 0,Y 425.318,Z 235.504,A -85,B 0,C 180,E1 -9961.367,E2 -9961.367} C_VEL
LIN {X 0,Y 425.277,Z 235.511,A -85,B 0,C 180,E1 -9964.553,E2 -9964.553} C_VEL
LIN {X 0,Y 425.289,Z 235.509,A -85,B 0,C 180,E1 -9966.634,E2 -9966.634} C_VEL
LIN {X 0,Y 425.3,Z 235.508,A -85,B 0,C 180,E1 -9969.694,E2 -9969.694} C_VEL
LIN {X 0,Y 425.337,Z 235.505,A -85,B 0,C 180,E1 -9972.697,E2 -9972.697} C_VEL
LIN {X 0,Y 425.35,Z 235.502,A -85,B 0,C 180,E1 -9975.65,E2 -9975.65} C_VEL
LIN {X 0,Y 425.353,Z 235.502,A -85,B 0,C 180,E1 -9978.564,E2 -9978.564} C_VEL
LIN {X 0,Y 425.41,Z 235.493,A -85,B 0,C 180,E1 -9981.449,E2 -9981.449} C_VEL
LIN {X 0,Y 425.508,Z 235.482,A -85,B 0,C 180,E1 -9984.312,E2 -9984.312} C_VEL
LIN {X 0,Y 425.567,Z 235.474,A -85,B 0,C 180,E1 -9988.107,E2 -9988.107} C_VEL
LIN {X 0,Y 425.615,Z 235.469,A -85,B 0,C 180,E1 -9990,E2 -9990} C_VEL
LIN {X 0,Y 425.534,Z 235.476,A -85,B 0,C 180,E1 -9992.84,E2 -9992.84} C_VEL
LIN {X 0,Y 425.297,Z 235.508,A -85,B 0,C 180,E1 -9993.759,E2 -9993.759} C_VEL
LIN {X 0,Y 424.51,Z 235.801,A -85,B 0,C 180,E1 -9994.546,E2 -9994.546} C_VEL
LIN {X 0,Y 421.57,Z 237.226,A -85,B 0,C 180,E1 -9995.813,E2 -9995.813} C_VEL
LIN {X 0,Y 419.139,Z 238.975,A -85,B 0,C 180,E1 -9996.825,E2 -9996.825} C_VEL
LIN {X 0,Y 418.096,Z 240.51,A -85,B 0,C 180,E1 -9997.6,E2 -9997.6} C_VEL
LIN {X 0,Y 418.008,Z 241.046,A -85,B 0,C 180,E1 -9997.862,E2 -9997.862} C_VEL
LIN {X 0,Y 417.913,Z 248.867,A -85,B 0,C 180,E1 -10001.642,E2 -10001.642} C_VEL
LIN {X 0,Y 417.778,Z 254.992,A -85,B 0,C 180,E1 -10004.616,E2 -10004.616} C_VEL
LIN {X 0,Y 417.673,Z 262.208,A -85,B 0,C 180,E1 -10008.137,E2 -10008.137} C_VEL
LIN {X 0,Y 417.524,Z 269.573,A -85,B 0,C 180,E1 -10011.735,E2 -10011.735} C_VEL
LIN {X 0,Y 417.536,Z 273.386,A -85,B 0,C 180,E1 -10013.596,E2 -10013.596} C_VEL
LIN {X 0,Y 419.941,Z 286.912,A -85,B 0,C 180,E1 -10014.206,E2 -10014.206} C_VEL
LIN {X 0,Y 420.181,Z 291.281,A -85,B 0,C 180,E1 -10014.455,E2 -10014.455} C_VEL
LIN {X 0,Y 419.823,Z 301.449,A -85,B 0,C 180,E1 -10015.107,E2 -10015.107} C_VEL
LIN {X 0,Y 419.401,Z 311.427,A -85,B 0,C 180,E1 -10015.962,E2 -10015.962} C_VEL
LIN {X 0,Y 418.999,Z 319.136,A -85,B 0,C 180,E1 -10016.794,E2 -10016.794} C_VEL
LIN {X 0,Y 418.642,Z 325.275,A -85,B 0,C 180,E1 -10017.585,E2 -10017.585} C_VEL
LIN {X 0,Y 418.285,Z 331.855,A -85,B 0,C 180,E1 -10018.611,E2 -10018.611} C_VEL
LIN {X 0,Y 418.02,Z 336.419,A -85,B 0,C 180,E1 -10019.457,E2 -10019.457} C_VEL
LIN {X 0,Y 417.734,Z 341.472,A -85,B 0,C 180,E1 -10020.597,E2 -10020.597} C_VEL
LIN {X 0,Y 417.55,Z 344.629,A -85,B 0,C 180,E1 -10021.452,E2 -10021.452} C_VEL
LIN {X 0,Y 417.346,Z 348.122,A -85,B 0,C 180,E1 -10022.649,E2 -10022.649} C_VEL
LIN {X 0,Y 417.208,Z 350.593,A -85,B 0,C 180,E1 -10023.772,E2 -10023.772} C_VEL
LIN {X 0,Y 417.089,Z 352.389,A -85,B 0,C 180,E1 -10024.953,E2 -10024.953} C_VEL
LIN {X 0,Y 417.039,Z 353.423,A -85,B 0,C 180,E1 -10026.145,E2 -10026.145} C_VEL
LIN {X 0,Y 417.01,Z 353.613,A -85,B 0,C 180,E1 -10027.617,E2 -10027.617} C_VEL
LIN {X 0,Y 417.1,Z 352.584,A -85,B 0,C 180,E1 -10029.187,E2 -10029.187} C_VEL
LIN {X 0,Y 417.301,Z 350.305,A -85,B 0,C 180,E1 -10030.723,E2 -10030.723} C_VEL
LIN {X 0,Y 417.549,Z 346.323,A -85,B 0,C 180,E1 -10032.319,E2 -10032.319} C_VEL
LIN {X 0,Y 417.766,Z 343.186,A -85,B 0,C 180,E1 -10033.277,E2 -10033.277} C_VEL
LIN {X 0,Y 418.053,Z 337.779,A -85,B 0,C 180,E1 -10034.577,E2 -10034.577} C_VEL
LIN {X 0,Y 418.43,Z 332.396,A -85,B 0,C 180,E1 -10035.614,E2 -10035.614} C_VEL
LIN {X 0,Y 418.839,Z 325.441,A -85,B 0,C 180,E1 -10036.711,E2 -10036.711} C_VEL
LIN {X 0,Y 419.398,Z 315.72,A -85,B 0,C 180,E1 -10037.91,E2 -10037.91} C_VEL
LIN {X 0,Y 419.867,Z 307.672,A -85,B 0,C 180,E1 -10038.688,E2 -10038.688} C_VEL
LIN {X 0,Y 420.262,Z 299.016,A -85,B 0,C 180,E1 -10039.362,E2 -10039.362} C_VEL
LIN {X 0,Y 420.497,Z 289.413,A -85,B 0,C 180,E1 -10039.948,E2 -10039.948} C_VEL
LIN {X 0,Y 418.423,Z 277.604,A -85,B 0,C 180,E1 -10040.544,E2 -10040.544} C_VEL
LIN {X 0,Y 417.661,Z 274.013,A -85,B 0,C 180,E1 -10040.707,E2 -10040.707} C_VEL
LIN {X 0,Y 417.71,Z 267.383,A -85,B 0,C 180,E1 -10043.922,E2 -10043.922} C_VEL
LIN {X 0,Y 417.846,Z 261.388,A -85,B 0,C 180,E1 -10046.809,E2 -10046.809} C_VEL
LIN {X 0,Y 417.906,Z 255.356,A -85,B 0,C 180,E1 -10049.701,E2 -10049.701} C_VEL
LIN {X 0,Y 417.999,Z 249.605,A -85,B 0,C 180,E1 -10052.46,E2 -10052.46} C_VEL
LIN {X 0,Y 418.144,Z 241.36,A -85,B 0,C 180,E1 -10056.21,E2 -10056.21} C_VEL
LIN {X 0,Y 418.16,Z 236.405,A -85,B 0,C 180,E1 -10058.558,E2 -10058.558} C_VEL
LIN {X 0,Y 418.283,Z 236.385,A -85,B 0,C 180,E1 -10061.383,E2 -10061.383} C_VEL
LIN {X 0,Y 418.305,Z 236.382,A -85,B 0,C 180,E1 -10064.406,E2 -10064.406} C_VEL
LIN {X 0,Y 418.358,Z 236.376,A -85,B 0,C 180,E1 -10067.386,E2 -10067.386} C_VEL
LIN {X 0,Y 418.344,Z 236.377,A -85,B 0,C 180,E1 -10070.329,E2 -10070.329} C_VEL
LIN {X 0,Y 418.448,Z 236.364,A -85,B 0,C 180,E1 -10073.248,E2 -10073.248} C_VEL
LIN {X 0,Y 418.337,Z 236.378,A -85,B 0,C 180,E1 -10075.181,E2 -10075.181} C_VEL
LIN {X 0,Y 418.545,Z 236.351,A -85,B 0,C 180,E1 -10078.075,E2 -10078.075} C_VEL
LIN {X 0,Y 418.674,Z 236.335,A -85,B 0,C 180,E1 -10080,E2 -10080} C_VEL
LIN {X 0,Y 418.503,Z 236.356,A -85,B 0,C 180,E1 -10082.888,E2 -10082.888} C_VEL
LIN {X 0,Y 418.501,Z 236.356,A -85,B 0,C 180,E1 -10085.783,E2 -10085.783} C_VEL
LIN {X 0,Y 418.399,Z 236.369,A -85,B 0,C 180,E1 -10088.695,E2 -10088.695} C_VEL
LIN {X 0,Y 418.317,Z 236.378,A -85,B 0,C 180,E1 -10091.631,E2 -10091.631} C_VEL
LIN {X 0,Y 418.306,Z 236.381,A -85,B 0,C 180,E1 -10094.597,E2 -10094.597} C_VEL
LIN {X 0,Y 418.288,Z 236.383,A -85,B 0,C 180,E1 -10097.604,E2 -10097.604} C_VEL
LIN {X 0,Y 418.252,Z 236.386,A -85,B 0,C 180,E1 -10100.663,E2 -10100.663} C_VEL
LIN {X 0,Y 418.275,Z 236.384,A -85,B 0,C 180,E1 -10103.782,E2 -10103.782} C_VEL
LIN {X 0,Y 418.312,Z 236.377,A -85,B 0,C 180,E1 -10107.07,E2 -10107.07} C_VEL
LIN {X 0,Y 418.246,Z 236.387,A -85,B 0,C 180,E1 -10110.272,E2 -10110.272} C_VEL
LIN {X 0,Y 418.249,Z 236.387,A -85,B 0,C 180,E1 -10113.677,E2 -10113.677} C_VEL
LIN {X 0,Y 418.242,Z 236.387,A -85,B 0,C 180,E1 -10117.224,E2 -10117.224} C_VEL
LIN {X 0,Y 418.253,Z 236.385,A -85,B 0,C 180,E1 -10119.682,E2 -10119.682} C_VEL
LIN {X 0,Y 418.231,Z 236.388,A -85,B 0,C 180,E1 -10122.321,E2 -10122.321} C_VEL
LIN {X 0,Y 418.237,Z 236.39,A -85,B 0,C 180,E1 -10125.109,E2 -10125.109} C_VEL
LIN {X 0,Y 418.298,Z 236.497,A -85,B 0,C 180,E1 -10127.936,E2 -10127.936} C_VEL
LIN {X 0,Y 419.391,Z 242.718,A -85,B 0,C 180,E1 -10131.093,E2 -10131.093} C_VEL
LIN {X 0,Y 420.117,Z 247.523,A -85,B 0,C 180,E1 -10133.416,E2 -10133.416} C_VEL
LIN {X 0,Y 419.974,Z 252.962,A -85,B 0,C 180,E1 -10135.903,E2 -10135.903} C_VEL
LIN {X 0,Y 419.401,Z 259.35,A -85,B 0,C 180,E1 -10138.718,E2 -10138.718} C_VEL
LIN {X 0,Y 418.814,Z 266.945,A -85,B 0,C 180,E1 -10141.975,E2 -10141.975} C_VEL
LIN {X 0,Y 418.372,Z 274.568,A -85,B 0,C 180,E1 -10145.168,E2 -10145.168} C_VEL
LIN {X 0,Y 417.971,Z 282.159,A -85,B 0,C 180,E1 -10148.289,E2 -10148.289} C_VEL
LIN {X 0,Y 417.627,Z 289.756,A -85,B 0,C 180,E1 -10151.353,E2 -10151.353} C_VEL
LIN {X 0,Y 417.516,Z 294.081,A -85,B 0,C 180,E1 -10153.089,E2 -10153.089} C_VEL
LIN {X 0,Y 419.38,Z 308.086,A -85,B 0,C 180,E1 -10153.627,E2 -10153.627} C_VEL
LIN {X 0,Y 420.785,Z 320.521,A -85,B 0,C 180,E1 -10154.283,E2 -10154.283} C_VEL
LIN {X 0,Y 420.496,Z 329.824,A -85,B 0,C 180,E1 -10154.862,E2 -10154.862} C_VEL
LIN {X 0,Y 419.752,Z 342.18,A -85,B 0,C 180,E1 -10155.826,E2 -10155.826} C_VEL
LIN {X 0,Y 419.089,Z 352.16,A -85,B 0,C 180,E1 -10156.795,E2 -10156.795} C_VEL
LIN {X 0,Y 418.577,Z 361.391,A -85,B 0,C 180,E1 -10157.885,E2 -10157.885} C_VEL
LIN {X 0,Y 418.057,Z 369.872,A -85,B 0,C 180,E1 -10159.098,E2 -10159.098} C_VEL
LIN {X 0,Y 417.633,Z 378.173,A -85,B 0,C 180,E1 -10160.557,E2 -10160.557} C_VEL
LIN {X 0,Y 417.373,Z 384.868,A -85,B 0,C 180,E1 -10162.015,E2 -10162.015} C_VEL
LIN {X 0,Y 417.152,Z 390.984,A -85,B 0,C 180,E1 -10163.726,E2 -10163.726} C_VEL
LIN {X 0,Y 417.15,Z 394.873,A -85,B 0,C 180,E1 -10165.168,E2 -10165.168} C_VEL
LIN {X 0,Y 417.058,Z 396.868,A -85,B 0,C 180,E1 -10166.135,E2 -10166.135} C_VEL
LIN {X 0,Y 417.174,Z 398.447,A -85,B 0,C 180,E1 -10167.103,E2 -10167.103} C_VEL
LIN {X 0,Y 417.132,Z 399.566,A -85,B 0,C 180,E1 -10168.069,E2 -10168.069} C_VEL
LIN {X 0,Y 417.12,Z 400.235,A -85,B 0,C 180,E1 -10169.035,E2 -10169.035} C_VEL
LIN {X 0,Y 417.121,Z 400.497,A -85,B 0,C 180,E1 -10170,E2 -10170} C_VEL
LIN {X 0,Y 417.094,Z 400.351,A -85,B 0,C 180,E1 -10170.966,E2 -10170.966} C_VEL
LIN {X 0,Y 417.122,Z 399.764,A -85,B 0,C 180,E1 -10171.931,E2 -10171.931} C_VEL
LIN {X 0,Y 417.124,Z 398.742,A -85,B 0,C 180,E1 -10172.897,E2 -10172.897} C_VEL
LIN {X 0,Y 417.051,Z 397.301,A -85,B 0,C 180,E1 -10173.865,E2 -10173.865} C_VEL
LIN {X 0,Y 417.14,Z 394.303,A -85,B 0,C 180,E1 -10175.317,E2 -10175.317} C_VEL
LIN {X 0,Y 417.231,Z 390.247,A -85,B 0,C 180,E1 -10176.772,E2 -10176.772} C_VEL
LIN {X 0,Y 417.446,Z 384.068,A -85,B 0,C 180,E1 -10178.471,E2 -10178.471} C_VEL
LIN {X 0,Y 417.801,Z 377.3,A -85,B 0,C 180,E1 -10179.929,E2 -10179.929} C_VEL
LIN {X 0,Y 418.368,Z 368.987,A -85,B 0,C 180,E1 -10181.384,E2 -10181.384} C_VEL
LIN {X 0,Y 418.978,Z 360.591,A -85,B 0,C 180,E1 -10182.596,E2 -10182.596} C_VEL
LIN {X 0,Y 419.612,Z 350.711,A -85,B 0,C 180,E1 -10183.783,E2 -10183.783} C_VEL
LIN {X 0,Y 420.578,Z 339.321,A -85,B 0,C 180,E1 -10184.888,E2 -10184.888} C_VEL
LIN {X 0,Y 421.506,Z 327.056,A -85,B 0,C 180,E1 -10185.845,E2 -10185.845} C_VEL
LIN {X 0,Y 421.649,Z 321.608,A -85,B 0,C 180,E1 -10186.212,E2 -10186.212} C_VEL
LIN {X 0,Y 420.64,Z 307.895,A -85,B 0,C 180,E1 -10187.039,E2 -10187.039} C_VEL
LIN {X 0,Y 418.259,Z 294.449,A -85,B 0,C 180,E1 -10187.739,E2 -10187.739} C_VEL
LIN {X 0,Y 417.512,Z 290.647,A -85,B 0,C 180,E1 -10187.923,E2 -10187.923} C_VEL
LIN {X 0,Y 417.868,Z 282.571,A -85,B 0,C 180,E1 -10191.199,E2 -10191.199} C_VEL
LIN {X 0,Y 418.214,Z 275.271,A -85,B 0,C 180,E1 -10194.313,E2 -10194.313} C_VEL
LIN {X 0,Y 418.698,Z 268.936,A -85,B 0,C 180,E1 -10197.174,E2 -10197.174} C_VEL
LIN {X 0,Y 419.276,Z 262.742,A -85,B 0,C 180,E1 -10200.19,E2 -10200.19} C_VEL
LIN {X 0,Y 420.143,Z 256.617,A -85,B 0,C 180,E1 -10203.506,E2 -10203.506} C_VEL
LIN {X 0,Y 420.577,Z 252.925,A -85,B 0,C 180,E1 -10205.794,E2 -10205.794} C_VEL
LIN {X 0,Y 420.515,Z 249.622,A -85,B 0,C 180,E1 -10208.233,E2 -10208.233} C_VEL
LIN {X 0,Y 420.04,Z 246.52,A -85,B 0,C 180,E1 -10211.155,E2 -10211.155} C_VEL
LIN {X 0,Y 419.676,Z 244.37,A -85,B 0,C 180,E1 -10213.938,E2 -10213.938} C_VEL
LIN {X 0,Y 419.405,Z 243.023,A -85,B 0,C 180,E1 -10216.604,E2 -10216.604} C_VEL
LIN {X 0,Y 419.276,Z 242.327,A -85,B 0,C 180,E1 -10219.177,E2 -10219.177} C_VEL
LIN {X 0,Y 419.205,Z 242.177,A -85,B 0,C 180,E1 -10221.996,E2 -10221.996} C_VEL
LIN {X 0,Y 419.098,Z 242.728,A -85,B 0,C 180,E1 -10225.256,E2 -10225.256} C_VEL
LIN {X 0,Y 418.862,Z 243.495,A -85,B 0,C 180,E1 -10227.526,E2 -10227.526} C_VEL
LIN {X 0,Y 418.527,Z 245.047,A -85,B 0,C 180,E1 -10230.858,E2 -10230.858} C_VEL
LIN {X 0,Y 418.26,Z 246.931,A -85,B 0,C 180,E1 -10234.095,E2 -10234.095} C_VEL
LIN {X 0,Y 418.036,Z 249.054,A -85,B 0,C 180,E1 -10237.252,E2 -10237.252} C_VEL
LIN {X 0,Y 417.918,Z 251.351,A -85,B 0,C 180,E1 -10240.346,E2 -10240.346} C_VEL
LIN {X 0,Y 417.803,Z 253.677,A -85,B 0,C 180,E1 -10243.242,E2 -10243.242} C_VEL
LIN {X 0,Y 422.041,Z 267.235,A -85,B 0,C 180,E1 -10244.114,E2 -10244.114} C_VEL
LIN {X 0,Y 423.332,Z 272.938,A -85,B 0,C 180,E1 -10244.504,E2 -10244.504} C_VEL
LIN {X 0,Y 422.637,Z 284.928,A -85,B 0,C 180,E1 -10245.262,E2 -10245.262} C_VEL
LIN {X 0,Y 421.79,Z 297.181,A -85,B 0,C 180,E1 -10246.265,E2 -10246.265} C_VEL
LIN {X 0,Y 420.916,Z 307.786,A -85,B 0,C 180,E1 -10247.341,E2 -10247.341} C_VEL
LIN {X 0,Y 420.236,Z 316.477,A -85,B 0,C 180,E1 -10248.423,E2 -10248.423} C_VEL
LIN {X 0,Y 419.423,Z 325.943,A -85,B 0,C 180,E1 -10249.867,E2 -10249.867} C_VEL
LIN {X 0,Y 418.748,Z 333.635,A -85,B 0,C 180,E1 -10251.312,E2 -10251.312} C_VEL
LIN {X 0,Y 418.167,Z 340.217,A -85,B 0,C 180,E1 -10252.878,E2 -10252.878} C_VEL
LIN {X 0,Y 417.874,Z 346.035,A -85,B 0,C 180,E1 -10254.693,E2 -10254.693} C_VEL
LIN {X 0,Y 417.707,Z 349.446,A -85,B 0,C 180,E1 -10256.141,E2 -10256.141} C_VEL
LIN {X 0,Y 417.535,Z 351.163,A -85,B 0,C 180,E1 -10257.106,E2 -10257.106} C_VEL
LIN {X 0,Y 417.21,Z 353.321,A -85,B 0,C 180,E1 -10259.035,E2 -10259.035} C_VEL
LIN {X 0,Y 417.176,Z 353.799,A -85,B 0,C 180,E1 -10260,E2 -10260} C_VEL
LIN {X 0,Y 417.143,Z 353.835,A -85,B 0,C 180,E1 -10260.965,E2 -10260.965} C_VEL
LIN {X 0,Y 417.259,Z 352.696,A -85,B 0,C 180,E1 -10262.897,E2 -10262.897} C_VEL
LIN {X 0,Y 417.255,Z 351.523,A -85,B 0,C 180,E1 -10263.863,E2 -10263.863} C_VEL
LIN {X 0,Y 417.338,Z 348.933,A -85,B 0,C 180,E1 -10265.315,E2 -10265.315} C_VEL
LIN {X 0,Y 417.481,Z 345.047,A -85,B 0,C 180,E1 -10266.857,E2 -10266.857} C_VEL
LIN {X 0,Y 417.703,Z 340.57,A -85,B 0,C 180,E1 -10268.223,E2 -10268.223} C_VEL
LIN {X 0,Y 418.049,Z 334.547,A -85,B 0,C 180,E1 -10269.678,E2 -10269.678} C_VEL
LIN {X 0,Y 418.45,Z 327.051,A -85,B 0,C 180,E1 -10271.137,E2 -10271.137} C_VEL
LIN {X 0,Y 419.099,Z 317.767,A -85,B 0,C 180,E1 -10272.592,E2 -10272.592} C_VEL
LIN {X 0,Y 419.608,Z 307.5,A -85,B 0,C 180,E1 -10273.884,E2 -10273.884} C_VEL
LIN {X 0,Y 420.285,Z 296.292,A -85,B 0,C 180,E1 -10275.022,E2 -10275.022} C_VEL
LIN {X 0,Y 421.023,Z 284.199,A -85,B 0,C 180,E1 -10275.988,E2 -10275.988} C_VEL
LIN {X 0,Y 421.562,Z 271.812,A -85,B 0,C 180,E1 -10276.763,E2 -10276.763} C_VEL
LIN {X 0,Y 420.276,Z 263.965,A -85,B 0,C 180,E1 -10277.197,E2 -10277.197} C_VEL
LIN {X 0,Y 417.352,Z 250.514,A -85,B 0,C 180,E1 -10277.806,E2 -10277.806} C_VEL
LIN {X 0,Y 417.261,Z 249.816,A -85,B 0,C 180,E1 -10277.839,E2 -10277.839} C_VEL
LIN {X 0,Y 417.284,Z 246.684,A -85,B 0,C 180,E1 -10280.713,E2 -10280.713} C_VEL
LIN {X 0,Y 417.353,Z 242.561,A -85,B 0,C 180,E1 -10284.586,E2 -10284.586} C_VEL
LIN {X 0,Y 417.448,Z 239.998,A -85,B 0,C 180,E1 -10287.037,E2 -10287.037} C_VEL
LIN {X 0,Y 417.473,Z 236.623,A -85,B 0,C 180,E1 -10290.334,E2 -10290.334} C_VEL
LIN {X 0,Y 417.864,Z 236.437,A -85,B 0,C 180,E1 -10293.713,E2 -10293.713} C_VEL
LIN {X 0,Y 418.157,Z 236.397,A -85,B 0,C 180,E1 -10296.221,E2 -10296.221} C_VEL
LIN {X 0,Y 418.244,Z 236.388,A -85,B 0,C 180,E1 -10299.378,E2 -10299.378} C_VEL
LIN {X 0,Y 418.227,Z 236.388,A -85,B 0,C 180,E1 -10302.32,E2 -10302.32} C_VEL
LIN {X 0,Y 418.239,Z 236.389,A -85,B 0,C 180,E1 -10305.109,E2 -10305.109} C_VEL
LIN {X 0,Y 418.226,Z 236.387,A -85,B 0,C 180,E1 -10307.765,E2 -10307.765} C_VEL
LIN {X 0,Y 418.236,Z 236.385,A -85,B 0,C 180,E1 -10311.556,E2 -10311.556} C_VEL
LIN {X 0,Y 418.252,Z 236.385,A -85,B 0,C 180,E1 -10315.158,E2 -10315.158} C_VEL
LIN {X 0,Y 418.247,Z 236.384,A -85,B 0,C 180,E1 -10317.472,E2 -10317.472} C_VEL
LIN {X 0,Y 418.268,Z 236.383,A -85,B 0,C 180,E1 -10320.897,E2 -10320.897} C_VEL
LIN {X 0,Y 418.242,Z 236.389,A -85,B 0,C 180,E1 -10324.094,E2 -10324.094} C_VEL
LIN {X 0,Y 418.236,Z 236.387,A -85,B 0,C 180,E1 -10327.263,E2 -10327.263} C_VEL
LIN {X 0,Y 418.287,Z 236.382,A -85,B 0,C 180,E1 -10330.364,E2 -10330.364} C_VEL
LIN {X 0,Y 418.32,Z 236.377,A -85,B 0,C 180,E1 -10333.404,E2 -10333.404} C_VEL
LIN {X 0,Y 418.35,Z 236.373,A -85,B 0,C 180,E1 -10336.999,E2 -10336.999} C_VEL
LIN {X 0,Y 418.339,Z 236.377,A -85,B 0,C 180,E1 -10340.328,E2 -10340.328} C_VEL
LIN {X 0,Y 418.441,Z 236.361,A -85,B 0,C 180,E1 -10343.248,E2 -10343.248} C_VEL
LIN {X 0,Y 418.313,Z 236.376,A -85,B 0,C 180,E1 -10345.181,E2 -10345.181} C_VEL
LIN {X 0,Y 418.536,Z 236.351,A -85,B 0,C 180,E1 -10348.075,E2 -10348.075} C_VEL
LIN {X 0,Y 418.567,Z 236.347,A -85,B 0,C 180,E1 -10350,E2 -10350} C_VEL
LIN {X 0,Y 418.488,Z 236.354,A -85,B 0,C 180,E1 -10352.888,E2 -10352.888} C_VEL
LIN {X 0,Y 418.13,Z 236.475,A -85,B 0,C 180,E1 -10355.667,E2 -10355.667} C_VEL
LIN {X 0,Y 418.008,Z 241.046,A -85,B 0,C 180,E1 -10357.862,E2 -10357.862} C_VEL
LIN {X 0,Y 417.324,Z 242.722,A -85,B 0,C 180,E1 -10358.633,E2 -10358.633} C_VEL
LIN {X 0,Y 414.435,Z 245.656,A -85,B 0,C 180,E1 -10359.875,E2 -10359.875} C_VEL
LIN {X 0,Y 411.997,Z 248.034,A -85,B 0,C 180,E1 -10360.877,E2 -10360.877} C_VEL
LIN {X 0,Y 410.952,Z 249.77,A -85,B 0,C 180,E1 -10361.656,E2 -10361.656} C_VEL
LIN {X 0,Y 410.868,Z 250.319,A -85,B 0,C 180,E1 -10361.92,E2 -10361.92} C_VEL
LIN {X 0,Y 410.729,Z 257.409,A -85,B 0,C 180,E1 -10365.38,E2 -10365.38} C_VEL
LIN {X 0,Y 410.611,Z 263.682,A -85,B 0,C 180,E1 -10368.46,E2 -10368.46} C_VEL
LIN {X 0,Y 410.465,Z 270.082,A -85,B 0,C 180,E1 -10371.6,E2 -10371.6} C_VEL
LIN {X 0,Y 410.461,Z 273.731,A -85,B 0,C 180,E1 -10373.392,E2 -10373.392} C_VEL
LIN {X 0,Y 412.642,Z 285.794,A -85,B 0,C 180,E1 -10373.927,E2 -10373.927} C_VEL
LIN {X 0,Y 413.272,Z 290.906,A -85,B 0,C 180,E1 -10374.221,E2 -10374.221} C_VEL
LIN {X 0,Y 412.949,Z 299.703,A -85,B 0,C 180,E1 -10374.777,E2 -10374.777} C_VEL
LIN {X 0,Y 412.514,Z 309.7,A -85,B 0,C 180,E1 -10375.588,E2 -10375.588} C_VEL
LIN {X 0,Y 412.016,Z 319.185,A -85,B 0,C 180,E1 -10376.6,E2 -10376.6} C_VEL
LIN {X 0,Y 411.64,Z 325.681,A -85,B 0,C 180,E1 -10377.45,E2 -10377.45} C_VEL
LIN {X 0,Y 411.35,Z 331.178,A -85,B 0,C 180,E1 -10378.302,E2 -10378.302} C_VEL
LIN {X 0,Y 410.947,Z 337.395,A -85,B 0,C 180,E1 -10379.477,E2 -10379.477} C_VEL
LIN {X 0,Y 410.648,Z 342.231,A -85,B 0,C 180,E1 -10380.608,E2 -10380.608} C_VEL
LIN {X 0,Y 410.45,Z 345.572,A -85,B 0,C 180,E1 -10381.562,E2 -10381.562} C_VEL
LIN {X 0,Y 410.253,Z 349.258,A -85,B 0,C 180,E1 -10382.921,E2 -10382.921} C_VEL
LIN {X 0,Y 410.04,Z 352.444,A -85,B 0,C 180,E1 -10384.642,E2 -10384.642} C_VEL
LIN {X 0,Y 409.942,Z 353.865,A -85,B 0,C 180,E1 -10386.315,E2 -10386.315} C_VEL
LIN {X 0,Y 409.94,Z 353.864,A -85,B 0,C 180,E1 -10388.111,E2 -10388.111} C_VEL
LIN {X 0,Y 410.057,Z 352.692,A -85,B 0,C 180,E1 -10389.532,E2 -10389.532} C_VEL
LIN {X 0,Y 410.282,Z 350.074,A -85,B 0,C 180,E1 -10391.087,E2 -10391.087} C_VEL
LIN {X 0,Y 410.48,Z 347.246,A -85,B 0,C 180,E1 -10392.249,E2 -10392.249} C_VEL
LIN {X 0,Y 410.766,Z 342.693,A -85,B 0,C 180,E1 -10393.638,E2 -10393.638} C_VEL
LIN {X 0,Y 411.131,Z 336.784,A -85,B 0,C 180,E1 -10395.025,E2 -10395.025} C_VEL
LIN {X 0,Y 411.631,Z 329.49,A -85,B 0,C 180,E1 -10396.344,E2 -10396.344} C_VEL
LIN {X 0,Y 412.128,Z 322.517,A -85,B 0,C 180,E1 -10397.342,E2 -10397.342} C_VEL
LIN {X 0,Y 412.472,Z 315.994,A -85,B 0,C 180,E1 -10398.123,E2 -10398.123} C_VEL
LIN {X 0,Y 412.932,Z 308.787,A -85,B 0,C 180,E1 -10398.839,E2 -10398.839} C_VEL
LIN {X 0,Y 413.322,Z 300.013,A -85,B 0,C 180,E1 -10399.545,E2 -10399.545} C_VEL
LIN {X 0,Y 413.655,Z 290.696,A -85,B 0,C 180,E1 -10400.131,E2 -10400.131} C_VEL
LIN {X 0,Y 411.688,Z 279.31,A -85,B 0,C 180,E1 -10400.742,E2 -10400.742} C_VEL
LIN {X 0,Y 410.605,Z 274.413,A -85,B 0,C 180,E1 -10400.943,E2 -10400.943} C_VEL
LIN {X 0,Y 410.7,Z 269.11,A -85,B 0,C 180,E1 -10403.541,E2 -10403.541} C_VEL
LIN {X 0,Y 410.806,Z 262.04,A -85,B 0,C 180,E1 -10406.96,E2 -10406.96} C_VEL
LIN {X 0,Y 410.92,Z 255.236,A -85,B 0,C 180,E1 -10410.265,E2 -10410.265} C_VEL
LIN {X 0,Y 410.969,Z 249.905,A -85,B 0,C 180,E1 -10412.78,E2 -10412.78} C_VEL
LIN {X 0,Y 411.155,Z 242.288,A -85,B 0,C 180,E1 -10416.316,E2 -10416.316} C_VEL
LIN {X 0,Y 411.125,Z 237.28,A -85,B 0,C 180,E1 -10418.699,E2 -10418.699} C_VEL
LIN {X 0,Y 411.222,Z 237.264,A -85,B 0,C 180,E1 -10421.051,E2 -10421.051} C_VEL
LIN {X 0,Y 411.257,Z 237.259,A -85,B 0,C 180,E1 -10424.132,E2 -10424.132} C_VEL
LIN {X 0,Y 411.306,Z 237.253,A -85,B 0,C 180,E1 -10427.166,E2 -10427.166} C_VEL
LIN {X 0,Y 411.296,Z 237.255,A -85,B 0,C 180,E1 -10430.161,E2 -10430.161} C_VEL
LIN {X 0,Y 411.396,Z 237.243,A -85,B 0,C 180,E1 -10433.132,E2 -10433.132} C_VEL
LIN {X 0,Y 411.308,Z 237.253,A -85,B 0,C 180,E1 -10435.099,E2 -10435.099} C_VEL
LIN {X 0,Y 411.514,Z 237.227,A -85,B 0,C 180,E1 -10438.042,E2 -10438.042} C_VEL
LIN {X 0,Y 411.643,Z 237.21,A -85,B 0,C 180,E1 -10440,E2 -10440} C_VEL
LIN {X 0,Y 411.459,Z 237.233,A -85,B 0,C 180,E1 -10442.937,E2 -10442.937} C_VEL
LIN {X 0,Y 411.426,Z 237.237,A -85,B 0,C 180,E1 -10446.867,E2 -10446.867} C_VEL
LIN {X 0,Y 411.295,Z 237.254,A -85,B 0,C 180,E1 -10449.839,E2 -10449.839} C_VEL
LIN {X 0,Y 411.308,Z 237.252,A -85,B 0,C 180,E1 -10453.104,E2 -10453.104} C_VEL
LIN {X 0,Y 411.265,Z 237.258,A -85,B 0,C 180,E1 -10456.869,E2 -10456.869} C_VEL
LIN {X 0,Y 411.233,Z 237.261,A -85,B 0,C 180,E1 -10459.987,E2 -10459.987} C_VEL
LIN {X 0,Y 411.197,Z 237.266,A -85,B 0,C 180,E1 -10463.148,E2 -10463.148} C_VEL
LIN {X 0,Y 411.235,Z 237.26,A -85,B 0,C 180,E1 -10466.381,E2 -10466.381} C_VEL
LIN {X 0,Y 411.202,Z 237.263,A -85,B 0,C 180,E1 -10469.713,E2 -10469.713} C_VEL
LIN {X 0,Y 411.208,Z 237.264,A -85,B 0,C 180,E1 -10473.156,E2 -10473.156} C_VEL
LIN {X 0,Y 411.194,Z 237.265,A -85,B 0,C 180,E1 -10476.552,E2 -10476.552} C_VEL
LIN {X 0,Y 411.217,Z 237.262,A -85,B 0,C 180,E1 -10479.728,E2 -10479.728} C_VEL
LIN {X 0,Y 411.174,Z 237.27,A -85,B 0,C 180,E1 -10483.134,E2 -10483.134} C_VEL
LIN {X 0,Y 411.169,Z 237.27,A -85,B 0,C 180,E1 -10485.881,E2 -10485.881} C_VEL
LIN {X 0,Y 411.249,Z 237.374,A -85,B 0,C 180,E1 -10487.701,E2 -10487.701} C_VEL
LIN {X 0,Y 412.321,Z 243.573,A -85,B 0,C 180,E1 -10490.901,E2 -10490.901} C_VEL
LIN {X 0,Y 413.103,Z 248.739,A -85,B 0,C 180,E1 -10493.456,E2 -10493.456} C_VEL
LIN {X 0,Y 412.976,Z 253.861,A -85,B 0,C 180,E1 -10495.834,E2 -10495.834} C_VEL
LIN {X 0,Y 412.411,Z 259.664,A -85,B 0,C 180,E1 -10498.437,E2 -10498.437} C_VEL
LIN {X 0,Y 411.876,Z 266.555,A -85,B 0,C 180,E1 -10501.46,E2 -10501.46} C_VEL
LIN {X 0,Y 411.326,Z 274.593,A -85,B 0,C 180,E1 -10504.9,E2 -10504.9} C_VEL
LIN {X 0,Y 410.92,Z 281.724,A -85,B 0,C 180,E1 -10507.897,E2 -10507.897} C_VEL
LIN {X 0,Y 410.575,Z 289.287,A -85,B 0,C 180,E1 -10511.02,E2 -10511.02} C_VEL
LIN {X 0,Y 410.438,Z 293.75,A -85,B 0,C 180,E1 -10512.846,E2 -10512.846} C_VEL
LIN {X 0,Y 412.423,Z 308.702,A -85,B 0,C 180,E1 -10513.455,E2 -10513.455} C_VEL
LIN {X 0,Y 413.776,Z 321.113,A -85,B 0,C 180,E1 -10514.135,E2 -10514.135} C_VEL
LIN {X 0,Y 413.485,Z 330.225,A -85,B 0,C 180,E1 -10514.725,E2 -10514.725} C_VEL
LIN {X 0,Y 412.726,Z 342.418,A -85,B 0,C 180,E1 -10515.705,E2 -10515.705} C_VEL
LIN {X 0,Y 412.03,Z 353.207,A -85,B 0,C 180,E1 -10516.795,E2 -10516.795} C_VEL
LIN {X 0,Y 411.392,Z 364.086,A -85,B 0,C 180,E1 -10518.17,E2 -10518.17} C_VEL
LIN {X 0,Y 410.843,Z 372.047,A -85,B 0,C 180,E1 -10519.404,E2 -10519.404} C_VEL
LIN {X 0,Y 410.438,Z 379.862,A -85,B 0,C 180,E1 -10520.887,E2 -10520.887} C_VEL
LIN {X 0,Y 410.267,Z 385.2,A -85,B 0,C 180,E1 -10522.123,E2 -10522.123} C_VEL
LIN {X 0,Y 410.073,Z 390.736,A -85,B 0,C 180,E1 -10523.736,E2 -10523.736} C_VEL
LIN {X 0,Y 410.081,Z 394.327,A -85,B 0,C 180,E1 -10525.084,E2 -10525.084} C_VEL
LIN {X 0,Y 409.974,Z 396.343,A -85,B 0,C 180,E1 -10526.068,E2 -10526.068} C_VEL
LIN {X 0,Y 410.086,Z 397.942,A -85,B 0,C 180,E1 -10527.053,E2 -10527.053} C_VEL
LIN {X 0,Y 410.059,Z 399.1,A -85,B 0,C 180,E1 -10528.036,E2 -10528.036} C_VEL
LIN {X 0,Y 410.039,Z 399.791,A -85,B 0,C 180,E1 -10529.018,E2 -10529.018} C_VEL
LIN {X 0,Y 410.037,Z 400.072,A -85,B 0,C 180,E1 -10530,E2 -10530} C_VEL
LIN {X 0,Y 410.015,Z 399.943,A -85,B 0,C 180,E1 -10530.982,E2 -10530.982} C_VEL
LIN {X 0,Y 410.048,Z 399.391,A -85,B 0,C 180,E1 -10531.965,E2 -10531.965} C_VEL
LIN {X 0,Y 410.021,Z 398.383,A -85,B 0,C 180,E1 -10532.948,E2 -10532.948} C_VEL
LIN {X 0,Y 409.968,Z 396.961,A -85,B 0,C 180,E1 -10533.932,E2 -10533.932} C_VEL
LIN {X 0,Y 410.032,Z 393.999,A -85,B 0,C 180,E1 -10535.41,E2 -10535.41} C_VEL
LIN {X 0,Y 410.163,Z 389.977,A -85,B 0,C 180,E1 -10536.889,E2 -10536.889} C_VEL
LIN {X 0,Y 410.341,Z 384.818,A -85,B 0,C 180,E1 -10538.371,E2 -10538.371} C_VEL
LIN {X 0,Y 410.704,Z 378.379,A -85,B 0,C 180,E1 -10539.853,E2 -10539.853} C_VEL
LIN {X 0,Y 411.236,Z 370.438,A -85,B 0,C 180,E1 -10541.335,E2 -10541.335} C_VEL
LIN {X 0,Y 412.032,Z 360.63,A -85,B 0,C 180,E1 -10542.811,E2 -10542.811} C_VEL
LIN {X 0,Y 412.716,Z 350.883,A -85,B 0,C 180,E1 -10544.018,E2 -10544.018} C_VEL
LIN {X 0,Y 413.754,Z 339.726,A -85,B 0,C 180,E1 -10545.139,E2 -10545.139} C_VEL
LIN {X 0,Y 414.725,Z 327.73,A -85,B 0,C 180,E1 -10546.111,E2 -10546.111} C_VEL
LIN {X 0,Y 414.856,Z 320.607,A -85,B 0,C 180,E1 -10546.612,E2 -10546.612} C_VEL
LIN {X 0,Y 413.939,Z 308.86,A -85,B 0,C 180,E1 -10547.356,E2 -10547.356} C_VEL
LIN {X 0,Y 411.68,Z 295.81,A -85,B 0,C 180,E1 -10548.08,E2 -10548.08} C_VEL
LIN {X 0,Y 410.484,Z 290.121,A -85,B 0,C 180,E1 -10548.369,E2 -10548.369} C_VEL
LIN {X 0,Y 410.856,Z 282.431,A -85,B 0,C 180,E1 -10551.579,E2 -10551.579} C_VEL
LIN {X 0,Y 411.342,Z 274.031,A -85,B 0,C 180,E1 -10555.286,E2 -10555.286} C_VEL
LIN {X 0,Y 411.929,Z 267.199,A -85,B 0,C 180,E1 -10558.537,E2 -10558.537} C_VEL
LIN {X 0,Y 412.717,Z 260.832,A -85,B 0,C 180,E1 -10561.863,E2 -10561.863} C_VEL
LIN {X 0,Y 413.306,Z 256.919,A -85,B 0,C 180,E1 -10564.135,E2 -10564.135} C_VEL
LIN {X 0,Y 413.658,Z 253.365,A -85,B 0,C 180,E1 -10566.488,E2 -10566.488} C_VEL
LIN {X 0,Y 413.445,Z 250.269,A -85,B 0,C 180,E1 -10568.973,E2 -10568.973} C_VEL
LIN {X 0,Y 413.039,Z 247.71,A -85,B 0,C 180,E1 -10571.575,E2 -10571.575} C_VEL
LIN {X 0,Y 412.688,Z 245.69,A -85,B 0,C 180,E1 -10574.336,E2 -10574.336} C_VEL
LIN {X 0,Y 412.447,Z 244.389,A -85,B 0,C 180,E1 -10577.115,E2 -10577.115} C_VEL
LIN {X 0,Y 412.275,Z 243.716,A -85,B 0,C 180,E1 -10580.096,E2 -10580.096} C_VEL
LIN {X 0,Y 412.249,Z 243.656,A -85,B 0,C 180,E1 -10582.141,E2 -10582.141} C_VEL
LIN {X 0,Y 412.132,Z 244.041,A -85,B 0,C 180,E1 -10584.939,E2 -10584.939} C_VEL
LIN {X 0,Y 411.957,Z 244.597,A -85,B 0,C 180,E1 -10586.912,E2 -10586.912} C_VEL
LIN {X 0,Y 411.604,Z 246.016,A -85,B 0,C 180,E1 -10590.319,E2 -10590.319} C_VEL
LIN {X 0,Y 411.285,Z 247.805,A -85,B 0,C 180,E1 -10593.622,E2 -10593.622} C_VEL
LIN {X 0,Y 411.052,Z 249.865,A -85,B 0,C 180,E1 -10596.843,E2 -10596.843} C_VEL
LIN {X 0,Y 410.902,Z 252.24,A -85,B 0,C 180,E1 -10600.173,E2 -10600.173} C_VEL
LIN {X 0,Y 410.768,Z 254.294,A -85,B 0,C 180,E1 -10602.802,E2 -10602.802} C_VEL
LIN {X 0,Y 415.085,Z 267.349,A -85,B 0,C 180,E1 -10603.684,E2 -10603.684} C_VEL
LIN {X 0,Y 416.733,Z 274.523,A -85,B 0,C 180,E1 -10604.198,E2 -10604.198} C_VEL
LIN {X 0,Y 415.903,Z 287.499,A -85,B 0,C 180,E1 -10605.071,E2 -10605.071} C_VEL
LIN {X 0,Y 415.035,Z 298.764,A -85,B 0,C 180,E1 -10606.037,E2 -10606.037} C_VEL
LIN {X 0,Y 414.105,Z 309.098,A -85,B 0,C 180,E1 -10607.129,E2 -10607.129} C_VEL
LIN {X 0,Y 413.254,Z 319.305,A -85,B 0,C 180,E1 -10608.473,E2 -10608.473} C_VEL
LIN {X 0,Y 412.415,Z 328.33,A -85,B 0,C 180,E1 -10609.941,E2 -10609.941} C_VEL
LIN {X 0,Y 411.736,Z 335.585,A -85,B 0,C 180,E1 -10611.411,E2 -10611.411} C_VEL
LIN {X 0,Y 411.005,Z 342.313,A -85,B 0,C 180,E1 -10613.125,E2 -10613.125} C_VEL
LIN {X 0,Y 410.85,Z 346.723,A -85,B 0,C 180,E1 -10614.602,E2 -10614.602} C_VEL
LIN {X 0,Y 410.662,Z 350.064,A -85,B 0,C 180,E1 -10616.075,E2 -10616.075} C_VEL
LIN {X 0,Y 410.495,Z 351.721,A -85,B 0,C 180,E1 -10617.056,E2 -10617.056} C_VEL
LIN {X 0,Y 410.157,Z 353.816,A -85,B 0,C 180,E1 -10619.018,E2 -10619.018} C_VEL
LIN {X 0,Y 410.089,Z 354.247,A -85,B 0,C 180,E1 -10620,E2 -10620} C_VEL
LIN {X 0,Y 410.061,Z 354.239,A -85,B 0,C 180,E1 -10620.982,E2 -10620.982} C_VEL
LIN {X 0,Y 410.192,Z 353.032,A -85,B 0,C 180,E1 -10622.946,E2 -10622.946} C_VEL
LIN {X 0,Y 410.162,Z 351.798,A -85,B 0,C 180,E1 -10623.93,E2 -10623.93} C_VEL
LIN {X 0,Y 410.281,Z 349.144,A -85,B 0,C 180,E1 -10625.406,E2 -10625.406} C_VEL
LIN {X 0,Y 410.397,Z 345.456,A -85,B 0,C 180,E1 -10626.885,E2 -10626.885} C_VEL
LIN {X 0,Y 410.646,Z 340.623,A -85,B 0,C 180,E1 -10628.365,E2 -10628.365} C_VEL
LIN {X 0,Y 411.009,Z 334.51,A -85,B 0,C 180,E1 -10629.846,E2 -10629.846} C_VEL
LIN {X 0,Y 411.456,Z 326.914,A -85,B 0,C 180,E1 -10631.328,E2 -10631.328} C_VEL
LIN {X 0,Y 412.021,Z 319.195,A -85,B 0,C 180,E1 -10632.561,E2 -10632.561} C_VEL
LIN {X 0,Y 412.467,Z 309.855,A -85,B 0,C 180,E1 -10633.801,E2 -10633.801} C_VEL
LIN {X 0,Y 413.213,Z 298.272,A -85,B 0,C 180,E1 -10635.033,E2 -10635.033} C_VEL
LIN {X 0,Y 413.945,Z 286.708,A -85,B 0,C 180,E1 -10636.016,E2 -10636.016} C_VEL
LIN {X 0,Y 414.512,Z 274.164,A -85,B 0,C 180,E1 -10636.846,E2 -10636.846} C_VEL
LIN {X 0,Y 414.379,Z 270.121,A -85,B 0,C 180,E1 -10637.079,E2 -10637.079} C_VEL
LIN {X 0,Y 411.554,Z 256.585,A -85,B 0,C 180,E1 -10637.792,E2 -10637.792} C_VEL
LIN {X 0,Y 410.222,Z 250.159,A -85,B 0,C 180,E1 -10638.059,E2 -10638.059} C_VEL
LIN {X 0,Y 410.193,Z 246.894,A -85,B 0,C 180,E1 -10641.088,E2 -10641.088} C_VEL
LIN {X 0,Y 410.306,Z 242.971,A -85,B 0,C 180,E1 -10644.793,E2 -10644.793} C_VEL
LIN {X 0,Y 410.353,Z 240.132,A -85,B 0,C 180,E1 -10647.544,E2 -10647.544} C_VEL
LIN {X 0,Y 410.4,Z 237.863,A -85,B 0,C 180,E1 -10649.777,E2 -10649.777} C_VEL
LIN {X 0,Y 410.51,Z 237.353,A -85,B 0,C 180,E1 -10651.128,E2 -10651.128} C_VEL
LIN {X 0,Y 410.895,Z 237.302,A -85,B 0,C 180,E1 -10654.363,E2 -10654.363} C_VEL
LIN {X 0,Y 411.153,Z 237.271,A -85,B 0,C 180,E1 -10656.746,E2 -10656.746} C_VEL
LIN {X 0,Y 411.21,Z 237.263,A -85,B 0,C 180,E1 -10659.727,E2 -10659.727} C_VEL
LIN {X 0,Y 411.175,Z 237.269,A -85,B 0,C 180,E1 -10663.134,E2 -10663.134} C_VEL
LIN {X 0,Y 411.168,Z 237.266,A -85,B 0,C 180,E1 -10665.881,E2 -10665.881} C_VEL
LIN {X 0,Y 411.152,Z 237.271,A -85,B 0,C 180,E1 -10668.774,E2 -10668.774} C_VEL
LIN {X 0,Y 411.184,Z 237.263,A -85,B 0,C 180,E1 -10672.025,E2 -10672.025} C_VEL
LIN {X 0,Y 411.204,Z 237.263,A -85,B 0,C 180,E1 -10675.124,E2 -10675.124} C_VEL
LIN {X 0,Y 411.168,Z 237.266,A -85,B 0,C 180,E1 -10678.003,E2 -10678.003} C_VEL
LIN {X 0,Y 411.205,Z 237.262,A -85,B 0,C 180,E1 -10681.409,E2 -10681.409} C_VEL
LIN {X 0,Y 411.23,Z 237.26,A -85,B 0,C 180,E1 -10684.929,E2 -10684.929} C_VEL
LIN {X 0,Y 411.208,Z 237.264,A -85,B 0,C 180,E1 -10687.913,E2 -10687.913} C_VEL
LIN {X 0,Y 411.223,Z 237.261,A -85,B 0,C 180,E1 -10691.051,E2 -10691.051} C_VEL
LIN {X 0,Y 411.258,Z 237.258,A -85,B 0,C 180,E1 -10694.132,E2 -10694.132} C_VEL
LIN {X 0,Y 411.307,Z 237.25,A -85,B 0,C 180,E1 -10697.166,E2 -10697.166} C_VEL
LIN {X 0,Y 411.292,Z 237.255,A -85,B 0,C 180,E1 -10700.161,E2 -10700.161} C_VEL
LIN {X 0,Y 411.391,Z 237.239,A -85,B 0,C 180,E1 -10703.132,E2 -10703.132} C_VEL
LIN {X 0,Y 411.285,Z 237.251,A -85,B 0,C 180,E1 -10705.099,E2 -10705.099} C_VEL
LIN {X 0,Y 411.505,Z 237.227,A -85,B 0,C 180,E1 -10708.042,E2 -10708.042} C_VEL
LIN {X 0,Y 411.519,Z 237.225,A -85,B 0,C 180,E1 -10710,E2 -10710} C_VEL
LIN {X 0,Y 411.443,Z 237.232,A -85,B 0,C 180,E1 -10712.937,E2 -10712.937} C_VEL
LIN {X 0,Y 411.096,Z 237.393,A -85,B 0,C 180,E1 -10715.641,E2 -10715.641} C_VEL
LIN {X 0,Y 410.911,Z 244.043,A -85,B 0,C 180,E1 -10718.855,E2 -10718.855} C_VEL
LIN {X 0,Y 410.868,Z 250.319,A -85,B 0,C 180,E1 -10721.92,E2 -10721.92} C_VEL
LIN {X 0,Y 410.184,Z 252.024,A -85,B 0,C 180,E1 -10722.703,E2 -10722.703} C_VEL
LIN {X 0,Y 407.253,Z 254.956,A -85,B 0,C 180,E1 -10723.967,E2 -10723.967} C_VEL
LIN {X 0,Y 404.78,Z 257.322,A -85,B 0,C 180,E1 -10724.987,E2 -10724.987} C_VEL
LIN {X 0,Y 403.729,Z 259.046,A -85,B 0,C 180,E1 -10725.78,E2 -10725.78} C_VEL
LIN {X 0,Y 403.65,Z 259.607,A -85,B 0,C 180,E1 -10726.049,E2 -10726.049} C_VEL
LIN {X 0,Y 403.535,Z 265.195,A -85,B 0,C 180,E1 -10728.796,E2 -10728.796} C_VEL
LIN {X 0,Y 403.425,Z 271.671,A -85,B 0,C 180,E1 -10731.996,E2 -10731.996} C_VEL
LIN {X 0,Y 403.419,Z 274.062,A -85,B 0,C 180,E1 -10733.179,E2 -10733.179} C_VEL
LIN {X 0,Y 405.343,Z 284.504,A -85,B 0,C 180,E1 -10733.638,E2 -10733.638} C_VEL
LIN {X 0,Y 406.31,Z 291.817,A -85,B 0,C 180,E1 -10734.052,E2 -10734.052} C_VEL
LIN {X 0,Y 405.94,Z 301.49,A -85,B 0,C 180,E1 -10734.688,E2 -10734.688} C_VEL
LIN {X 0,Y 405.414,Z 312.449,A -85,B 0,C 180,E1 -10735.651,E2 -10735.651} C_VEL
LIN {X 0,Y 404.982,Z 320.359,A -85,B 0,C 180,E1 -10736.543,E2 -10736.543} C_VEL
LIN {X 0,Y 404.612,Z 326.296,A -85,B 0,C 180,E1 -10737.341,E2 -10737.341} C_VEL
LIN {X 0,Y 404.273,Z 332.136,A -85,B 0,C 180,E1 -10738.276,E2 -10738.276} C_VEL
LIN {X 0,Y 403.99,Z 336.777,A -85,B 0,C 180,E1 -10739.15,E2 -10739.15} C_VEL
LIN {X 0,Y 403.657,Z 341.891,A -85,B 0,C 180,E1 -10740.326,E2 -10740.326} C_VEL
LIN {X 0,Y 403.374,Z 346.028,A -85,B 0,C 180,E1 -10741.513,E2 -10741.513} C_VEL
LIN {X 0,Y 403.2,Z 349.268,A -85,B 0,C 180,E1 -10742.707,E2 -10742.707} C_VEL
LIN {X 0,Y 403.05,Z 351.704,A -85,B 0,C 180,E1 -10743.917,E2 -10743.917} C_VEL
LIN {X 0,Y 402.918,Z 353.37,A -85,B 0,C 180,E1 -10745.142,E2 -10745.142} C_VEL
LIN {X 0,Y 402.851,Z 354.355,A -85,B 0,C 180,E1 -10746.63,E2 -10746.63} C_VEL
LIN {X 0,Y 402.885,Z 354.213,A -85,B 0,C 180,E1 -10748.28,E2 -10748.28} C_VEL
LIN {X 0,Y 403.039,Z 352.217,A -85,B 0,C 180,E1 -10750.18,E2 -10750.18} C_VEL
LIN {X 0,Y 403.261,Z 349.807,A -85,B 0,C 180,E1 -10751.473,E2 -10751.473} C_VEL
LIN {X 0,Y 403.523,Z 346.386,A -85,B 0,C 180,E1 -10752.785,E2 -10752.785} C_VEL
LIN {X 0,Y 403.82,Z 341.8,A -85,B 0,C 180,E1 -10754.119,E2 -10754.119} C_VEL
LIN {X 0,Y 404.243,Z 335.817,A -85,B 0,C 180,E1 -10755.464,E2 -10755.464} C_VEL
LIN {X 0,Y 404.688,Z 329.451,A -85,B 0,C 180,E1 -10756.588,E2 -10756.588} C_VEL
LIN {X 0,Y 405.179,Z 322.997,A -85,B 0,C 180,E1 -10757.527,E2 -10757.527} C_VEL
LIN {X 0,Y 405.586,Z 316.173,A -85,B 0,C 180,E1 -10758.355,E2 -10758.355} C_VEL
LIN {X 0,Y 406.054,Z 308.459,A -85,B 0,C 180,E1 -10759.126,E2 -10759.126} C_VEL
LIN {X 0,Y 406.445,Z 300.528,A -85,B 0,C 180,E1 -10759.772,E2 -10759.772} C_VEL
LIN {X 0,Y 406.785,Z 291.654,A -85,B 0,C 180,E1 -10760.344,E2 -10760.344} C_VEL
LIN {X 0,Y 405.075,Z 281.662,A -85,B 0,C 180,E1 -10760.908,E2 -10760.908} C_VEL
LIN {X 0,Y 403.566,Z 274.784,A -85,B 0,C 180,E1 -10761.21,E2 -10761.21} C_VEL
LIN {X 0,Y 403.636,Z 268.456,A -85,B 0,C 180,E1 -10764.318,E2 -10764.318} C_VEL
LIN {X 0,Y 403.82,Z 262.231,A -85,B 0,C 180,E1 -10767.349,E2 -10767.349} C_VEL
LIN {X 0,Y 403.931,Z 255.106,A -85,B 0,C 180,E1 -10770.845,E2 -10770.845} C_VEL
LIN {X 0,Y 403.986,Z 249.174,A -85,B 0,C 180,E1 -10773.665,E2 -10773.665} C_VEL
LIN {X 0,Y 404.161,Z 243.207,A -85,B 0,C 180,E1 -10776.425,E2 -10776.425} C_VEL
LIN {X 0,Y 404.102,Z 238.154,A -85,B 0,C 180,E1 -10778.846,E2 -10778.846} C_VEL
LIN {X 0,Y 404.21,Z 238.138,A -85,B 0,C 180,E1 -10781.762,E2 -10781.762} C_VEL
LIN {X 0,Y 404.209,Z 238.136,A -85,B 0,C 180,E1 -10784.882,E2 -10784.882} C_VEL
LIN {X 0,Y 404.26,Z 238.132,A -85,B 0,C 180,E1 -10787.958,E2 -10787.958} C_VEL
LIN {X 0,Y 404.292,Z 238.126,A -85,B 0,C 180,E1 -10790.999,E2 -10790.999} C_VEL
LIN {X 0,Y 404.386,Z 238.115,A -85,B 0,C 180,E1 -10794.014,E2 -10794.014} C_VEL
LIN {X 0,Y 404.483,Z 238.103,A -85,B 0,C 180,E1 -10798.008,E2 -10798.008} C_VEL
LIN {X 0,Y 404.612,Z 238.086,A -85,B 0,C 180,E1 -10800,E2 -10800} C_VEL
LIN {X 0,Y 404.417,Z 238.11,A -85,B 0,C 180,E1 -10802.988,E2 -10802.988} C_VEL
LIN {X 0,Y 404.372,Z 238.116,A -85,B 0,C 180,E1 -10806.988,E2 -10806.988} C_VEL
LIN {X 0,Y 404.26,Z 238.13,A -85,B 0,C 180,E1 -10810.012,E2 -10810.012} C_VEL
LIN {X 0,Y 404.269,Z 238.128,A -85,B 0,C 180,E1 -10813.211,E2 -10813.211} C_VEL
LIN {X 0,Y 404.218,Z 238.136,A -85,B 0,C 180,E1 -10817.007,E2 -10817.007} C_VEL
LIN {X 0,Y 404.166,Z 238.143,A -85,B 0,C 180,E1 -10820.351,E2 -10820.351} C_VEL
LIN {X 0,Y 404.161,Z 238.142,A -85,B 0,C 180,E1 -10823.575,E2 -10823.575} C_VEL
LIN {X 0,Y 404.183,Z 238.139,A -85,B 0,C 180,E1 -10825.766,E2 -10825.766} C_VEL
LIN {X 0,Y 404.197,Z 238.137,A -85,B 0,C 180,E1 -10828,E2 -10828} C_VEL
LIN {X 0,Y 404.141,Z 238.143,A -85,B 0,C 180,E1 -10831.558,E2 -10831.558} C_VEL
LIN {X 0,Y 404.185,Z 238.138,A -85,B 0,C 180,E1 -10835.016,E2 -10835.016} C_VEL
LIN {X 0,Y 404.157,Z 238.142,A -85,B 0,C 180,E1 -10838.757,E2 -10838.757} C_VEL
LIN {X 0,Y 404.125,Z 238.147,A -85,B 0,C 180,E1 -10841.6,E2 -10841.6} C_VEL
LIN {X 0,Y 404.146,Z 238.145,A -85,B 0,C 180,E1 -10844.522,E2 -10844.522} C_VEL
LIN {X 0,Y 404.157,Z 238.197,A -85,B 0,C 180,E1 -10847.437,E2 -10847.437} C_VEL
LIN {X 0,Y 405.259,Z 244.417,A -85,B 0,C 180,E1 -10850.714,E2 -10850.714} C_VEL
LIN {X 0,Y 406.111,Z 249.718,A -85,B 0,C 180,E1 -10853.38,E2 -10853.38} C_VEL
LIN {X 0,Y 405.967,Z 254.715,A -85,B 0,C 180,E1 -10855.753,E2 -10855.753} C_VEL
LIN {X 0,Y 405.308,Z 261.075,A -85,B 0,C 180,E1 -10858.654,E2 -10858.654} C_VEL
LIN {X 0,Y 404.67,Z 269.355,A -85,B 0,C 180,E1 -10862.342,E2 -10862.342} C_VEL
LIN {X 0,Y 404.099,Z 277.499,A -85,B 0,C 180,E1 -10865.876,E2 -10865.876} C_VEL
LIN {X 0,Y 403.713,Z 285.048,A -85,B 0,C 180,E1 -10869.092,E2 -10869.092} C_VEL
LIN {X 0,Y 403.358,Z 293.412,A -85,B 0,C 180,E1 -10872.607,E2 -10872.607} C_VEL
LIN {X 0,Y 405.396,Z 309.113,A -85,B 0,C 180,E1 -10873.272,E2 -10873.272} C_VEL
LIN {X 0,Y 406.825,Z 322.167,A -85,B 0,C 180,E1 -10874.019,E2 -10874.019} C_VEL
LIN {X 0,Y 406.475,Z 330.527,A -85,B 0,C 180,E1 -10874.583,E2 -10874.583} C_VEL
LIN {X 0,Y 405.702,Z 342.577,A -85,B 0,C 180,E1 -10875.581,E2 -10875.581} C_VEL
LIN {X 0,Y 404.999,Z 352.768,A -85,B 0,C 180,E1 -10876.634,E2 -10876.634} C_VEL
LIN {X 0,Y 404.359,Z 363.147,A -85,B 0,C 180,E1 -10877.962,E2 -10877.962} C_VEL
LIN {X 0,Y 403.799,Z 371.198,A -85,B 0,C 180,E1 -10879.216,E2 -10879.216} C_VEL
LIN {X 0,Y 403.406,Z 379.128,A -85,B 0,C 180,E1 -10880.726,E2 -10880.726} C_VEL
LIN {X 0,Y 403.208,Z 384.509,A -85,B 0,C 180,E1 -10881.985,E2 -10881.985} C_VEL
LIN {X 0,Y 402.979,Z 390.531,A -85,B 0,C 180,E1 -10883.768,E2 -10883.768} C_VEL
LIN {X 0,Y 402.949,Z 394.834,A -85,B 0,C 180,E1 -10885.499,E2 -10885.499} C_VEL
LIN {X 0,Y 403,Z 397.427,A -85,B 0,C 180,E1 -10887.001,E2 -10887.001} C_VEL
LIN {X 0,Y 402.988,Z 398.617,A -85,B 0,C 180,E1 -10888.001,E2 -10888.001} C_VEL
LIN {X 0,Y 402.96,Z 399.343,A -85,B 0,C 180,E1 -10889.001,E2 -10889.001} C_VEL
LIN {X 0,Y 402.956,Z 399.643,A -85,B 0,C 180,E1 -10890,E2 -10890} C_VEL
LIN {X 0,Y 402.938,Z 399.534,A -85,B 0,C 180,E1 -10891,E2 -10891} C_VEL
LIN {X 0,Y 402.976,Z 399.016,A -85,B 0,C 180,E1 -10891.999,E2 -10891.999} C_VEL
LIN {X 0,Y 402.92,Z 398.032,A -85,B 0,C 180,E1 -10893,E2 -10893} C_VEL
LIN {X 0,Y 402.887,Z 396.628,A -85,B 0,C 180,E1 -10894.001,E2 -10894.001} C_VEL
LIN {X 0,Y 402.926,Z 393.709,A -85,B 0,C 180,E1 -10895.505,E2 -10895.505} C_VEL
LIN {X 0,Y 403.075,Z 389.737,A -85,B 0,C 180,E1 -10897.011,E2 -10897.011} C_VEL
LIN {X 0,Y 403.287,Z 384.624,A -85,B 0,C 180,E1 -10898.519,E2 -10898.519} C_VEL
LIN {X 0,Y 403.667,Z 378.255,A -85,B 0,C 180,E1 -10900.027,E2 -10900.027} C_VEL
LIN {X 0,Y 404.27,Z 370.415,A -85,B 0,C 180,E1 -10901.533,E2 -10901.533} C_VEL
LIN {X 0,Y 405.097,Z 360.732,A -85,B 0,C 180,E1 -10903.035,E2 -10903.035} C_VEL
LIN {X 0,Y 405.763,Z 351.976,A -85,B 0,C 180,E1 -10904.161,E2 -10904.161} C_VEL
LIN {X 0,Y 406.932,Z 340.233,A -85,B 0,C 180,E1 -10905.399,E2 -10905.399} C_VEL
LIN {X 0,Y 407.964,Z 328.526,A -85,B 0,C 180,E1 -10906.385,E2 -10906.385} C_VEL
LIN {X 0,Y 408.121,Z 321.643,A -85,B 0,C 180,E1 -10906.894,E2 -10906.894} C_VEL
LIN {X 0,Y 407.305,Z 309.979,A -85,B 0,C 180,E1 -10907.68,E2 -10907.68} C_VEL
LIN {X 0,Y 405.178,Z 297.495,A -85,B 0,C 180,E1 -10908.425,E2 -10908.425} C_VEL
LIN {X 0,Y 403.478,Z 289.529,A -85,B 0,C 180,E1 -10908.865,E2 -10908.865} C_VEL
LIN {X 0,Y 403.843,Z 282.303,A -85,B 0,C 180,E1 -10911.973,E2 -10911.973} C_VEL
LIN {X 0,Y 404.393,Z 274.016,A -85,B 0,C 180,E1 -10915.752,E2 -10915.752} C_VEL
LIN {X 0,Y 405.016,Z 267.304,A -85,B 0,C 180,E1 -10919.07,E2 -10919.07} C_VEL
LIN {X 0,Y 405.863,Z 261.072,A -85,B 0,C 180,E1 -10922.467,E2 -10922.467} C_VEL
LIN {X 0,Y 406.458,Z 257.281,A -85,B 0,C 180,E1 -10924.792,E2 -10924.792} C_VEL
LIN {X 0,Y 406.693,Z 253.691,A -85,B 0,C 180,E1 -10927.352,E2 -10927.352} C_VEL
LIN {X 0,Y 406.392,Z 250.929,A -85,B 0,C 180,E1 -10929.782,E2 -10929.782} C_VEL
LIN {X 0,Y 405.975,Z 248.545,A -85,B 0,C 180,E1 -10932.466,E2 -10932.466} C_VEL
LIN {X 0,Y 405.658,Z 246.753,A -85,B 0,C 180,E1 -10935.262,E2 -10935.262} C_VEL
LIN {X 0,Y 405.465,Z 245.599,A -85,B 0,C 180,E1 -10938.188,E2 -10938.188} C_VEL
LIN {X 0,Y 405.321,Z 245.131,A -85,B 0,C 180,E1 -10941.375,E2 -10941.375} C_VEL
LIN {X 0,Y 405.197,Z 245.371,A -85,B 0,C 180,E1 -10944.608,E2 -10944.608} C_VEL
LIN {X 0,Y 404.921,Z 246.132,A -85,B 0,C 180,E1 -10947.449,E2 -10947.449} C_VEL
LIN {X 0,Y 404.555,Z 247.561,A -85,B 0,C 180,E1 -10950.894,E2 -10950.894} C_VEL
LIN {X 0,Y 404.232,Z 249.355,A -85,B 0,C 180,E1 -10954.237,E2 -10954.237} C_VEL
LIN {X 0,Y 404.006,Z 251.413,A -85,B 0,C 180,E1 -10957.499,E2 -10957.499} C_VEL
LIN {X 0,Y 403.822,Z 253.678,A -85,B 0,C 180,E1 -10960.691,E2 -10960.691} C_VEL
LIN {X 0,Y 403.78,Z 255.027,A -85,B 0,C 180,E1 -10962.324,E2 -10962.324} C_VEL
LIN {X 0,Y 408.238,Z 268.016,A -85,B 0,C 180,E1 -10963.261,E2 -10963.261} C_VEL
LIN {X 0,Y 410.186,Z 276.541,A -85,B 0,C 180,E1 -10963.905,E2 -10963.905} C_VEL
LIN {X 0,Y 409.257,Z 289.19,A -85,B 0,C 180,E1 -10964.797,E2 -10964.797} C_VEL
LIN {X 0,Y 408.292,Z 300.429,A -85,B 0,C 180,E1 -10965.801,E2 -10965.801} C_VEL
LIN {X 0,Y 407.213,Z 311.478,A -85,B 0,C 180,E1 -10967.035,E2 -10967.035} C_VEL
LIN {X 0,Y 406.394,Z 320.499,A -85,B 0,C 180,E1 -10968.276,E2 -10968.276} C_VEL
LIN {X 0,Y 405.499,Z 329.342,A -85,B 0,C 180,E1 -10969.767,E2 -10969.767} C_VEL
LIN {X 0,Y 404.786,Z 336.48,A -85,B 0,C 180,E1 -10971.262,E2 -10971.262} C_VEL
LIN {X 0,Y 404.112,Z 342.246,A -85,B 0,C 180,E1 -10972.757,E2 -10972.757} C_VEL
LIN {X 0,Y 403.829,Z 347.416,A -85,B 0,C 180,E1 -10974.507,E2 -10974.507} C_VEL
LIN {X 0,Y 403.606,Z 350.685,A -85,B 0,C 180,E1 -10976.006,E2 -10976.006} C_VEL
LIN {X 0,Y 403.455,Z 352.294,A -85,B 0,C 180,E1 -10977.005,E2 -10977.005} C_VEL
LIN {X 0,Y 403.219,Z 353.509,A -85,B 0,C 180,E1 -10978.002,E2 -10978.002} C_VEL
LIN {X 0,Y 403.088,Z 354.32,A -85,B 0,C 180,E1 -10979.001,E2 -10979.001} C_VEL
LIN {X 0,Y 403.006,Z 354.687,A -85,B 0,C 180,E1 -10980,E2 -10980} C_VEL
LIN {X 0,Y 403.026,Z 354.201,A -85,B 0,C 180,E1 -10981.999,E2 -10981.999} C_VEL
LIN {X 0,Y 403.126,Z 353.357,A -85,B 0,C 180,E1 -10982.998,E2 -10982.998} C_VEL
LIN {X 0,Y 403.071,Z 352.064,A -85,B 0,C 180,E1 -10983.999,E2 -10983.999} C_VEL
LIN {X 0,Y 403.225,Z 349.333,A -85,B 0,C 180,E1 -10985.501,E2 -10985.501} C_VEL
LIN {X 0,Y 403.346,Z 345.562,A -85,B 0,C 180,E1 -10987.006,E2 -10987.006} C_VEL
LIN {X 0,Y 403.608,Z 340.642,A -85,B 0,C 180,E1 -10988.512,E2 -10988.512} C_VEL
LIN {X 0,Y 403.962,Z 334.436,A -85,B 0,C 180,E1 -10990.019,E2 -10990.019} C_VEL
LIN {X 0,Y 404.44,Z 326.737,A -85,B 0,C 180,E1 -10991.528,E2 -10991.528} C_VEL
LIN {X 0,Y 405.046,Z 318.903,A -85,B 0,C 180,E1 -10992.781,E2 -10992.781} C_VEL
LIN {X 0,Y 405.532,Z 309.371,A -85,B 0,C 180,E1 -10994.042,E2 -10994.042} C_VEL
LIN {X 0,Y 406.214,Z 298.905,A -85,B 0,C 180,E1 -10995.17,E2 -10995.17} C_VEL
LIN {X 0,Y 406.966,Z 287.442,A -85,B 0,C 180,E1 -10996.169,E2 -10996.169} C_VEL
LIN {X 0,Y 407.567,Z 274.483,A -85,B 0,C 180,E1 -10997.046,E2 -10997.046} C_VEL
LIN {X 0,Y 407.368,Z 270.927,A -85,B 0,C 180,E1 -10997.26,E2 -10997.26} C_VEL
LIN {X 0,Y 404.376,Z 256.539,A -85,B 0,C 180,E1 -10998.032,E2 -10998.032} C_VEL
LIN {X 0,Y 403.117,Z 250.502,A -85,B 0,C 180,E1 -10998.289,E2 -10998.289} C_VEL
LIN {X 0,Y 403.106,Z 247.089,A -85,B 0,C 180,E1 -11001.477,E2 -11001.477} C_VEL
LIN {X 0,Y 403.262,Z 243.385,A -85,B 0,C 180,E1 -11005.007,E2 -11005.007} C_VEL
LIN {X 0,Y 403.309,Z 240.252,A -85,B 0,C 180,E1 -11008.067,E2 -11008.067} C_VEL
LIN {X 0,Y 403.35,Z 238.244,A -85,B 0,C 180,E1 -11010.351,E2 -11010.351} C_VEL
LIN {X 0,Y 403.794,Z 238.188,A -85,B 0,C 180,E1 -11013.846,E2 -11013.846} C_VEL
LIN {X 0,Y 404.103,Z 238.15,A -85,B 0,C 180,E1 -11016.868,E2 -11016.868} C_VEL
LIN {X 0,Y 404.151,Z 238.141,A -85,B 0,C 180,E1 -11020.08,E2 -11020.08} C_VEL
LIN {X 0,Y 404.154,Z 238.143,A -85,B 0,C 180,E1 -11023.083,E2 -11023.083} C_VEL
LIN {X 0,Y 404.149,Z 238.141,A -85,B 0,C 180,E1 -11025.926,E2 -11025.926} C_VEL
LIN {X 0,Y 404.107,Z 238.148,A -85,B 0,C 180,E1 -11028.633,E2 -11028.633} C_VEL
LIN {X 0,Y 404.14,Z 238.141,A -85,B 0,C 180,E1 -11031.495,E2 -11031.495} C_VEL
LIN {X 0,Y 404.175,Z 238.14,A -85,B 0,C 180,E1 -11034.982,E2 -11034.982} C_VEL
LIN {X 0,Y 404.142,Z 238.145,A -85,B 0,C 180,E1 -11038.442,E2 -11038.442} C_VEL
LIN {X 0,Y 404.171,Z 238.139,A -85,B 0,C 180,E1 -11041.998,E2 -11041.998} C_VEL
LIN {X 0,Y 404.168,Z 238.139,A -85,B 0,C 180,E1 -11045.333,E2 -11045.333} C_VEL
LIN {X 0,Y 404.142,Z 238.144,A -85,B 0,C 180,E1 -11048.581,E2 -11048.581} C_VEL
LIN {X 0,Y 404.208,Z 238.136,A -85,B 0,C 180,E1 -11051.762,E2 -11051.762} C_VEL
LIN {X 0,Y 404.209,Z 238.134,A -85,B 0,C 180,E1 -11054.882,E2 -11054.882} C_VEL
LIN {X 0,Y 404.259,Z 238.129,A -85,B 0,C 180,E1 -11057.958,E2 -11057.958} C_VEL
LIN {X 0,Y 404.268,Z 238.126,A -85,B 0,C 180,E1 -11060.998,E2 -11060.998} C_VEL
LIN {X 0,Y 404.366,Z 238.119,A -85,B 0,C 180,E1 -11064.014,E2 -11064.014} C_VEL
LIN {X 0,Y 404.473,Z 238.103,A -85,B 0,C 180,E1 -11068.008,E2 -11068.008} C_VEL
LIN {X 0,Y 404.354,Z 238.114,A -85,B 0,C 180,E1 -11070.996,E2 -11070.996} C_VEL
LIN {X 0,Y 404.399,Z 238.11,A -85,B 0,C 180,E1 -11072.988,E2 -11072.988} C_VEL
LIN {X 0,Y 404.076,Z 238.336,A -85,B 0,C 180,E1 -11075.614,E2 -11075.614} C_VEL
LIN {X 0,Y 403.882,Z 245.32,A -85,B 0,C 180,E1 -11079.01,E2 -11079.01} C_VEL
LIN {X 0,Y 403.833,Z 251.515,A -85,B 0,C 180,E1 -11082.054,E2 -11082.054} C_VEL
LIN {X 0,Y 403.67,Z 257.758,A -85,B 0,C 180,E1 -11085.138,E2 -11085.138} C_VEL
LIN {X 0,Y 403.65,Z 259.607,A -85,B 0,C 180,E1 -11086.049,E2 -11086.049} C_VEL
LIN {X 0,Y 402.982,Z 261.32,A -85,B 0,C 180,E1 -11086.846,E2 -11086.846} C_VEL
LIN {X 0,Y 400.053,Z 264.25,A -85,B 0,C 180,E1 -11088.132,E2 -11088.132} C_VEL
LIN {X 0,Y 397.562,Z 266.628,A -85,B 0,C 180,E1 -11089.17,E2 -11089.17} C_VEL
LIN {X 0,Y 396.49,Z 268.358,A -85,B 0,C 180,E1 -11089.977,E2 -11089.977} C_VEL
LIN {X 0,Y 396.403,Z 268.925,A -85,B 0,C 180,E1 -11090.252,E2 -11090.252} C_VEL
LIN {X 0,Y 396.378,Z 274.475,A -85,B 0,C 180,E1 -11092.959,E2 -11092.959} C_VEL
LIN {X 0,Y 398.132,Z 283.964,A -85,B 0,C 180,E1 -11093.374,E2 -11093.374} C_VEL
LIN {X 0,Y 399.367,Z 292.699,A -85,B 0,C 180,E1 -11093.875,E2 -11093.875} C_VEL
LIN {X 0,Y 398.94,Z 303.239,A -85,B 0,C 180,E1 -11094.595,E2 -11094.595} C_VEL
LIN {X 0,Y 398.406,Z 313.512,A -85,B 0,C 180,E1 -11095.547,E2 -11095.547} C_VEL
LIN {X 0,Y 397.997,Z 320.417,A -85,B 0,C 180,E1 -11096.338,E2 -11096.338} C_VEL
LIN {X 0,Y 397.548,Z 327.788,A -85,B 0,C 180,E1 -11097.364,E2 -11097.364} C_VEL
LIN {X 0,Y 397.163,Z 333.624,A -85,B 0,C 180,E1 -11098.346,E2 -11098.346} C_VEL
LIN {X 0,Y 396.804,Z 338.994,A -85,B 0,C 180,E1 -11099.439,E2 -11099.439} C_VEL
LIN {X 0,Y 396.426,Z 344.889,A -85,B 0,C 180,E1 -11100.939,E2 -11100.939} C_VEL
LIN {X 0,Y 396.2,Z 348.494,A -85,B 0,C 180,E1 -11102.151,E2 -11102.151} C_VEL
LIN {X 0,Y 396.023,Z 351.444,A -85,B 0,C 180,E1 -11103.479,E2 -11103.479} C_VEL
LIN {X 0,Y 395.876,Z 353.236,A -85,B 0,C 180,E1 -11104.618,E2 -11104.618} C_VEL
LIN {X 0,Y 395.794,Z 354.448,A -85,B 0,C 180,E1 -11105.872,E2 -11105.872} C_VEL
LIN {X 0,Y 395.773,Z 354.894,A -85,B 0,C 180,E1 -11107.14,E2 -11107.14} C_VEL
LIN {X 0,Y 395.813,Z 354.408,A -85,B 0,C 180,E1 -11108.624,E2 -11108.624} C_VEL
LIN {X 0,Y 395.965,Z 352.613,A -85,B 0,C 180,E1 -11110.252,E2 -11110.252} C_VEL
LIN {X 0,Y 396.122,Z 351.37,A -85,B 0,C 180,E1 -11111.03,E2 -11111.03} C_VEL
LIN {X 0,Y 396.377,Z 348.358,A -85,B 0,C 180,E1 -11112.358,E2 -11112.358} C_VEL
LIN {X 0,Y 396.655,Z 344.211,A -85,B 0,C 180,E1 -11113.71,E2 -11113.71} C_VEL
LIN {X 0,Y 397.06,Z 338.791,A -85,B 0,C 180,E1 -11115.073,E2 -11115.073} C_VEL
LIN {X 0,Y 397.598,Z 331.87,A -85,B 0,C 180,E1 -11116.446,E2 -11116.446} C_VEL
LIN {X 0,Y 398.209,Z 324.038,A -85,B 0,C 180,E1 -11117.651,E2 -11117.651} C_VEL
LIN {X 0,Y 398.637,Z 317.038,A -85,B 0,C 180,E1 -11118.527,E2 -11118.527} C_VEL
LIN {X 0,Y 399.164,Z 308.993,A -85,B 0,C 180,E1 -11119.348,E2 -11119.348} C_VEL
LIN {X 0,Y 399.604,Z 300.307,A -85,B 0,C 180,E1 -11120.063,E2 -11120.063} C_VEL
LIN {X 0,Y 399.863,Z 292.365,A -85,B 0,C 180,E1 -11120.585,E2 -11120.585} C_VEL
LIN {X 0,Y 398.276,Z 282.917,A -85,B 0,C 180,E1 -11121.135,E2 -11121.135} C_VEL
LIN {X 0,Y 396.547,Z 275.139,A -85,B 0,C 180,E1 -11121.495,E2 -11121.495} C_VEL
LIN {X 0,Y 396.629,Z 268.859,A -85,B 0,C 180,E1 -11124.596,E2 -11124.596} C_VEL
LIN {X 0,Y 396.794,Z 262.128,A -85,B 0,C 180,E1 -11127.902,E2 -11127.902} C_VEL
LIN {X 0,Y 396.91,Z 256.031,A -85,B 0,C 180,E1 -11130.86,E2 -11130.86} C_VEL
LIN {X 0,Y 396.972,Z 250.171,A -85,B 0,C 180,E1 -11133.73,E2 -11133.73} C_VEL
LIN {X 0,Y 397.137,Z 242.97,A -85,B 0,C 180,E1 -11137.087,E2 -11137.087} C_VEL
LIN {X 0,Y 397.074,Z 239.029,A -85,B 0,C 180,E1 -11138.997,E2 -11138.997} C_VEL
LIN {X 0,Y 397.176,Z 239.014,A -85,B 0,C 180,E1 -11142.493,E2 -11142.493} C_VEL
LIN {X 0,Y 397.179,Z 239.013,A -85,B 0,C 180,E1 -11145.657,E2 -11145.657} C_VEL
LIN {X 0,Y 397.202,Z 239.011,A -85,B 0,C 180,E1 -11148.777,E2 -11148.777} C_VEL
LIN {X 0,Y 397.311,Z 238.996,A -85,B 0,C 180,E1 -11152.131,E2 -11152.131} C_VEL
LIN {X 0,Y 397.247,Z 239.004,A -85,B 0,C 180,E1 -11154.925,E2 -11154.925} C_VEL
LIN {X 0,Y 397.452,Z 238.979,A -85,B 0,C 180,E1 -11157.973,E2 -11157.973} C_VEL
LIN {X 0,Y 397.582,Z 238.962,A -85,B 0,C 180,E1 -11160,E2 -11160} C_VEL
LIN {X 0,Y 397.377,Z 238.987,A -85,B 0,C 180,E1 -11163.041,E2 -11163.041} C_VEL
LIN {X 0,Y 397.347,Z 238.99,A -85,B 0,C 180,E1 -11166.092,E2 -11166.092} C_VEL
LIN {X 0,Y 397.254,Z 239.002,A -85,B 0,C 180,E1 -11169.162,E2 -11169.162} C_VEL
LIN {X 0,Y 397.221,Z 239.007,A -85,B 0,C 180,E1 -11172.258,E2 -11172.258} C_VEL
LIN {X 0,Y 397.182,Z 239.012,A -85,B 0,C 180,E1 -11175.392,E2 -11175.392} C_VEL
LIN {X 0,Y 397.163,Z 239.011,A -85,B 0,C 180,E1 -11178.573,E2 -11178.573} C_VEL
LIN {X 0,Y 397.098,Z 239.022,A -85,B 0,C 180,E1 -11181.818,E2 -11181.818} C_VEL
LIN {X 0,Y 397.152,Z 239.015,A -85,B 0,C 180,E1 -11185.512,E2 -11185.512} C_VEL
LIN {X 0,Y 397.124,Z 239.02,A -85,B 0,C 180,E1 -11188.544,E2 -11188.544} C_VEL
LIN {X 0,Y 397.08,Z 239.022,A -85,B 0,C 180,E1 -11192.072,E2 -11192.072} C_VEL
LIN {X 0,Y 397.12,Z 239.018,A -85,B 0,C 180,E1 -11195.503,E2 -11195.503} C_VEL
LIN {X 0,Y 397.132,Z 239.017,A -85,B 0,C 180,E1 -11198.862,E2 -11198.862} C_VEL
LIN {X 0,Y 397.07,Z 239.024,A -85,B 0,C 180,E1 -11202.267,E2 -11202.267} C_VEL
LIN {X 0,Y 397.088,Z 239.025,A -85,B 0,C 180,E1 -11205.069,E2 -11205.069} C_VEL
LIN {X 0,Y 397.15,Z 239.111,A -85,B 0,C 180,E1 -11207.228,E2 -11207.228} C_VEL
LIN {X 0,Y 398.219,Z 245.308,A -85,B 0,C 180,E1 -11210.554,E2 -11210.554} C_VEL
LIN {X 0,Y 399.065,Z 250.492,A -85,B 0,C 180,E1 -11213.217,E2 -11213.217} C_VEL
LIN {X 0,Y 398.944,Z 255.599,A -85,B 0,C 180,E1 -11215.686,E2 -11215.686} C_VEL
LIN {X 0,Y 398.262,Z 261.927,A -85,B 0,C 180,E1 -11218.629,E2 -11218.629} C_VEL
LIN {X 0,Y 397.631,Z 269.548,A -85,B 0,C 180,E1 -11222.096,E2 -11222.096} C_VEL
LIN {X 0,Y 397.116,Z 277.041,A -85,B 0,C 180,E1 -11225.424,E2 -11225.424} C_VEL
LIN {X 0,Y 396.666,Z 284.56,A -85,B 0,C 180,E1 -11228.702,E2 -11228.702} C_VEL
LIN {X 0,Y 396.287,Z 292.663,A -85,B 0,C 180,E1 -11232.186,E2 -11232.186} C_VEL
LIN {X 0,Y 396.282,Z 293.135,A -85,B 0,C 180,E1 -11232.386,E2 -11232.386} C_VEL
LIN {X 0,Y 398.186,Z 308.126,A -85,B 0,C 180,E1 -11233.02,E2 -11233.02} C_VEL
LIN {X 0,Y 399.692,Z 321.434,A -85,B 0,C 180,E1 -11233.791,E2 -11233.791} C_VEL
LIN {X 0,Y 399.75,Z 327.286,A -85,B 0,C 180,E1 -11234.187,E2 -11234.187} C_VEL
LIN {X 0,Y 398.924,Z 338.496,A -85,B 0,C 180,E1 -11235.069,E2 -11235.069} C_VEL
LIN {X 0,Y 398.114,Z 349.964,A -85,B 0,C 180,E1 -11236.21,E2 -11236.21} C_VEL
LIN {X 0,Y 397.44,Z 360.349,A -85,B 0,C 180,E1 -11237.49,E2 -11237.49} C_VEL
LIN {X 0,Y 396.925,Z 368.806,A -85,B 0,C 180,E1 -11238.769,E2 -11238.769} C_VEL
LIN {X 0,Y 396.418,Z 377.081,A -85,B 0,C 180,E1 -11240.304,E2 -11240.304} C_VEL
LIN {X 0,Y 396.16,Z 383.763,A -85,B 0,C 180,E1 -11241.841,E2 -11241.841} C_VEL
LIN {X 0,Y 395.955,Z 389.068,A -85,B 0,C 180,E1 -11243.376,E2 -11243.376} C_VEL
LIN {X 0,Y 395.921,Z 393.162,A -85,B 0,C 180,E1 -11244.908,E2 -11244.908} C_VEL
LIN {X 0,Y 395.82,Z 395.252,A -85,B 0,C 180,E1 -11245.927,E2 -11245.927} C_VEL
LIN {X 0,Y 395.902,Z 396.899,A -85,B 0,C 180,E1 -11246.947,E2 -11246.947} C_VEL
LIN {X 0,Y 395.919,Z 398.117,A -85,B 0,C 180,E1 -11247.966,E2 -11247.966} C_VEL
LIN {X 0,Y 395.885,Z 398.89,A -85,B 0,C 180,E1 -11248.983,E2 -11248.983} C_VEL
LIN {X 0,Y 395.878,Z 399.212,A -85,B 0,C 180,E1 -11250,E2 -11250} C_VEL
LIN {X 0,Y 395.863,Z 399.125,A -85,B 0,C 180,E1 -11251.017,E2 -11251.017} C_VEL
LIN {X 0,Y 395.904,Z 398.632,A -85,B 0,C 180,E1 -11252.035,E2 -11252.035} C_VEL
LIN {X 0,Y 395.819,Z 397.691,A -85,B 0,C 180,E1 -11253.054,E2 -11253.054} C_VEL
LIN {X 0,Y 395.807,Z 396.308,A -85,B 0,C 180,E1 -11254.073,E2 -11254.073} C_VEL
LIN {X 0,Y 395.831,Z 392.966,A -85,B 0,C 180,E1 -11255.812,E2 -11255.812} C_VEL
LIN {X 0,Y 396.055,Z 387.989,A -85,B 0,C 180,E1 -11257.648,E2 -11257.648} C_VEL
LIN {X 0,Y 396.405,Z 381.482,A -85,B 0,C 180,E1 -11259.439,E2 -11259.439} C_VEL
LIN {X 0,Y 396.882,Z 374.493,A -85,B 0,C 180,E1 -11260.974,E2 -11260.974} C_VEL
LIN {X 0,Y 397.749,Z 365.922,A -85,B 0,C 180,E1 -11262.501,E2 -11262.501} C_VEL
LIN {X 0,Y 398.42,Z 356.682,A -85,B 0,C 180,E1 -11263.856,E2 -11263.856} C_VEL
LIN {X 0,Y 399.604,Z 345.677,A -85,B 0,C 180,E1 -11265.166,E2 -11265.166} C_VEL
LIN {X 0,Y 400.805,Z 333.964,A -85,B 0,C 180,E1 -11266.294,E2 -11266.294} C_VEL
LIN {X 0,Y 401.468,Z 324.53,A -85,B 0,C 180,E1 -11267.051,E2 -11267.051} C_VEL
LIN {X 0,Y 400.775,Z 311.905,A -85,B 0,C 180,E1 -11267.961,E2 -11267.961} C_VEL
LIN {X 0,Y 398.665,Z 298.659,A -85,B 0,C 180,E1 -11268.813,E2 -11268.813} C_VEL
LIN {X 0,Y 396.473,Z 288.987,A -85,B 0,C 180,E1 -11269.379,E2 -11269.379} C_VEL
LIN {X 0,Y 396.904,Z 280.938,A -85,B 0,C 180,E1 -11272.961,E2 -11272.961} C_VEL
LIN {X 0,Y 397.461,Z 274.034,A -85,B 0,C 180,E1 -11276.236,E2 -11276.236} C_VEL
LIN {X 0,Y 398.111,Z 267.427,A -85,B 0,C 180,E1 -11279.624,E2 -11279.624} C_VEL
LIN {X 0,Y 399.051,Z 261.355,A -85,B 0,C 180,E1 -11283.091,E2 -11283.091} C_VEL
LIN {X 0,Y 399.604,Z 257.677,A -85,B 0,C 180,E1 -11285.478,E2 -11285.478} C_VEL
LIN {X 0,Y 399.665,Z 254.413,A -85,B 0,C 180,E1 -11287.986,E2 -11287.986} C_VEL
LIN {X 0,Y 399.299,Z 251.479,A -85,B 0,C 180,E1 -11290.814,E2 -11290.814} C_VEL
LIN {X 0,Y 398.942,Z 249.188,A -85,B 0,C 180,E1 -11293.757,E2 -11293.757} C_VEL
LIN {X 0,Y 398.636,Z 247.714,A -85,B 0,C 180,E1 -11296.562,E2 -11296.562} C_VEL
LIN {X 0,Y 398.433,Z 246.879,A -85,B 0,C 180,E1 -11299.331,E2 -11299.331} C_VEL
LIN {X 0,Y 398.323,Z 246.612,A -85,B 0,C 180,E1 -11302.56,E2 -11302.56} C_VEL
LIN {X 0,Y 398.158,Z 246.99,A -85,B 0,C 180,E1 -11305.609,E2 -11305.609} C_VEL
LIN {X 0,Y 397.89,Z 247.671,A -85,B 0,C 180,E1 -11308.002,E2 -11308.002} C_VEL
LIN {X 0,Y 397.487,Z 249.112,A -85,B 0,C 180,E1 -11311.485,E2 -11311.485} C_VEL
LIN {X 0,Y 397.198,Z 250.908,A -85,B 0,C 180,E1 -11314.871,E2 -11314.871} C_VEL
LIN {X 0,Y 396.933,Z 252.99,A -85,B 0,C 180,E1 -11318.172,E2 -11318.172} C_VEL
LIN {X 0,Y 396.772,Z 255.526,A -85,B 0,C 180,E1 -11321.769,E2 -11321.769} C_VEL
LIN {X 0,Y 401.705,Z 269.613,A -85,B 0,C 180,E1 -11322.883,E2 -11322.883} C_VEL
LIN {X 0,Y 403.568,Z 277.492,A -85,B 0,C 180,E1 -11323.516,E2 -11323.516} C_VEL
LIN {X 0,Y 402.717,Z 289.747,A -85,B 0,C 180,E1 -11324.413,E2 -11324.413} C_VEL
LIN {X 0,Y 401.7,Z 300.935,A -85,B 0,C 180,E1 -11325.434,E2 -11325.434} C_VEL
LIN {X 0,Y 400.626,Z 310.937,A -85,B 0,C 180,E1 -11326.559,E2 -11326.559} C_VEL
LIN {X 0,Y 399.725,Z 320.084,A -85,B 0,C 180,E1 -11327.82,E2 -11327.82} C_VEL
LIN {X 0,Y 398.738,Z 329.109,A -85,B 0,C 180,E1 -11329.335,E2 -11329.335} C_VEL
LIN {X 0,Y 397.91,Z 336.351,A -85,B 0,C 180,E1 -11330.854,E2 -11330.854} C_VEL
LIN {X 0,Y 397.178,Z 342.598,A -85,B 0,C 180,E1 -11332.487,E2 -11332.487} C_VEL
LIN {X 0,Y 396.945,Z 346.819,A -85,B 0,C 180,E1 -11333.902,E2 -11333.902} C_VEL
LIN {X 0,Y 396.676,Z 350.349,A -85,B 0,C 180,E1 -11335.427,E2 -11335.427} C_VEL
LIN {X 0,Y 396.416,Z 352.883,A -85,B 0,C 180,E1 -11336.951,E2 -11336.951} C_VEL
LIN {X 0,Y 396.158,Z 354.06,A -85,B 0,C 180,E1 -11337.967,E2 -11337.967} C_VEL
LIN {X 0,Y 396.008,Z 354.817,A -85,B 0,C 180,E1 -11338.983,E2 -11338.983} C_VEL
LIN {X 0,Y 395.925,Z 355.129,A -85,B 0,C 180,E1 -11340,E2 -11340} C_VEL
LIN {X 0,Y 395.959,Z 354.565,A -85,B 0,C 180,E1 -11342.034,E2 -11342.034} C_VEL
LIN {X 0,Y 396.042,Z 353.656,A -85,B 0,C 180,E1 -11343.052,E2 -11343.052} C_VEL
LIN {X 0,Y 395.984,Z 352.316,A -85,B 0,C 180,E1 -11344.071,E2 -11344.071} C_VEL
LIN {X 0,Y 396.148,Z 349.505,A -85,B 0,C 180,E1 -11345.6,E2 -11345.6} C_VEL
LIN {X 0,Y 396.292,Z 345.649,A -85,B 0,C 180,E1 -11347.131,E2 -11347.131} C_VEL
LIN {X 0,Y 396.56,Z 340.639,A -85,B 0,C 180,E1 -11348.664,E2 -11348.664} C_VEL
LIN {X 0,Y 396.937,Z 334.337,A -85,B 0,C 180,E1 -11350.198,E2 -11350.198} C_VEL
LIN {X 0,Y 397.45,Z 326.518,A -85,B 0,C 180,E1 -11351.733,E2 -11351.733} C_VEL
LIN {X 0,Y 398.151,Z 316.736,A -85,B 0,C 180,E1 -11353.266,E2 -11353.266} C_VEL
LIN {X 0,Y 398.749,Z 306.705,A -85,B 0,C 180,E1 -11354.546,E2 -11354.546} C_VEL
LIN {X 0,Y 399.507,Z 295.49,A -85,B 0,C 180,E1 -11355.693,E2 -11355.693} C_VEL
LIN {X 0,Y 400.279,Z 283.03,A -85,B 0,C 180,E1 -11356.709,E2 -11356.709} C_VEL
LIN {X 0,Y 400.64,Z 273.133,A -85,B 0,C 180,E1 -11357.35,E2 -11357.35} C_VEL
LIN {X 0,Y 397.956,Z 259.972,A -85,B 0,C 180,E1 -11358.106,E2 -11358.106} C_VEL
LIN {X 0,Y 396.056,Z 250.828,A -85,B 0,C 180,E1 -11358.535,E2 -11358.535} C_VEL
LIN {X 0,Y 396.051,Z 247.276,A -85,B 0,C 180,E1 -11361.879,E2 -11361.879} C_VEL
LIN {X 0,Y 396.212,Z 243.801,A -85,B 0,C 180,E1 -11365.224,E2 -11365.224} C_VEL
LIN {X 0,Y 396.254,Z 240.365,A -85,B 0,C 180,E1 -11368.612,E2 -11368.612} C_VEL
LIN {X 0,Y 396.244,Z 239.21,A -85,B 0,C 180,E1 -11369.777,E2 -11369.777} C_VEL
LIN {X 0,Y 396.71,Z 239.072,A -85,B 0,C 180,E1 -11373.312,E2 -11373.312} C_VEL
LIN {X 0,Y 396.975,Z 239.037,A -85,B 0,C 180,E1 -11375.749,E2 -11375.749} C_VEL
LIN {X 0,Y 397.125,Z 239.019,A -85,B 0,C 180,E1 -11378.86,E2 -11378.86} C_VEL
LIN {X 0,Y 397.068,Z 239.023,A -85,B 0,C 180,E1 -11382.268,E2 -11382.268} C_VEL
LIN {X 0,Y 397.09,Z 239.024,A -85,B 0,C 180,E1 -11385.069,E2 -11385.069} C_VEL
LIN {X 0,Y 397.057,Z 239.024,A -85,B 0,C 180,E1 -11388.023,E2 -11388.023} C_VEL
LIN {X 0,Y 397.092,Z 239.019,A -85,B 0,C 180,E1 -11391.723,E2 -11391.723} C_VEL
LIN {X 0,Y 397.119,Z 239.015,A -85,B 0,C 180,E1 -11395.506,E2 -11395.506} C_VEL
LIN {X 0,Y 397.081,Z 239.022,A -85,B 0,C 180,E1 -11399.117,E2 -11399.117} C_VEL
LIN {X 0,Y 397.141,Z 239.016,A -85,B 0,C 180,E1 -11402.606,E2 -11402.606} C_VEL
LIN {X 0,Y 397.127,Z 239.018,A -85,B 0,C 180,E1 -11405.981,E2 -11405.981} C_VEL
LIN {X 0,Y 397.143,Z 239.015,A -85,B 0,C 180,E1 -11409.704,E2 -11409.704} C_VEL
LIN {X 0,Y 397.186,Z 239.01,A -85,B 0,C 180,E1 -11412.845,E2 -11412.845} C_VEL
LIN {X 0,Y 397.233,Z 239.004,A -85,B 0,C 180,E1 -11416.703,E2 -11416.703} C_VEL
LIN {X 0,Y 397.218,Z 239.006,A -85,B 0,C 180,E1 -11419.809,E2 -11419.809} C_VEL
LIN {X 0,Y 397.294,Z 238.994,A -85,B 0,C 180,E1 -11422.887,E2 -11422.887} C_VEL
LIN {X 0,Y 397.227,Z 239.002,A -85,B 0,C 180,E1 -11424.925,E2 -11424.925} C_VEL
LIN {X 0,Y 397.441,Z 238.979,A -85,B 0,C 180,E1 -11427.973,E2 -11427.973} C_VEL
LIN {X 0,Y 397.325,Z 238.99,A -85,B 0,C 180,E1 -11431.013,E2 -11431.013} C_VEL
LIN {X 0,Y 397.33,Z 238.99,A -85,B 0,C 180,E1 -11433.042,E2 -11433.042} C_VEL
LIN {X 0,Y 397.052,Z 239.153,A -85,B 0,C 180,E1 -11435.523,E2 -11435.523} C_VEL
LIN {X 0,Y 396.877,Z 245.577,A -85,B 0,C 180,E1 -11438.657,E2 -11438.657} C_VEL
LIN {X 0,Y 396.785,Z 252.862,A -85,B 0,C 180,E1 -11442.272,E2 -11442.272} C_VEL
LIN {X 0,Y 396.612,Z 260.267,A -85,B 0,C 180,E1 -11445.942,E2 -11445.942} C_VEL
LIN {X 0,Y 396.449,Z 266.703,A -85,B 0,C 180,E1 -11449.145,E2 -11449.145} C_VEL
LIN {X 0,Y 396.403,Z 268.925,A -85,B 0,C 180,E1 -11450.252,E2 -11450.252} C_VEL
LIN {X 0,Y 395.833,Z 271.042,A -85,B 0,C 180,E1 -11451.009,E2 -11451.009} C_VEL
LIN {X 0,Y 394.548,Z 273.987,A -85,B 0,C 180,E1 -11451.694,E2 -11451.694} C_VEL
LIN {X 0,Y 392.649,Z 278.952,A -85,B 0,C 180,E1 -11452.489,E2 -11452.489} C_VEL
LIN {X 0,Y 391.707,Z 283.397,A -85,B 0,C 180,E1 -11452.985,E2 -11452.985} C_VEL
LIN {X 0,Y 391.605,Z 286.663,A -85,B 0,C 180,E1 -11453.257,E2 -11453.257} C_VEL
LIN {X 0,Y 391.781,Z 288.367,A -85,B 0,C 180,E1 -11453.369,E2 -11453.369} C_VEL
LIN {X 0,Y 392.411,Z 292.327,A -85,B 0,C 180,E1 -11453.624,E2 -11453.624} C_VEL
LIN {X 0,Y 392.09,Z 301.19,A -85,B 0,C 180,E1 -11454.22,E2 -11454.22} C_VEL
LIN {X 0,Y 391.603,Z 311.244,A -85,B 0,C 180,E1 -11455.087,E2 -11455.087} C_VEL
LIN {X 0,Y 391.048,Z 320.295,A -85,B 0,C 180,E1 -11456.109,E2 -11456.109} C_VEL
LIN {X 0,Y 390.628,Z 326.89,A -85,B 0,C 180,E1 -11457.019,E2 -11457.019} C_VEL
LIN {X 0,Y 390.216,Z 333.111,A -85,B 0,C 180,E1 -11458.052,E2 -11458.052} C_VEL
LIN {X 0,Y 389.851,Z 338.47,A -85,B 0,C 180,E1 -11459.127,E2 -11459.127} C_VEL
LIN {X 0,Y 389.423,Z 344.539,A -85,B 0,C 180,E1 -11460.653,E2 -11460.653} C_VEL
LIN {X 0,Y 389.09,Z 349.43,A -85,B 0,C 180,E1 -11462.325,E2 -11462.325} C_VEL
LIN {X 0,Y 388.839,Z 352.823,A -85,B 0,C 180,E1 -11464.077,E2 -11464.077} C_VEL
LIN {X 0,Y 388.723,Z 354.543,A -85,B 0,C 180,E1 -11465.552,E2 -11465.552} C_VEL
LIN {X 0,Y 388.708,Z 355.276,A -85,B 0,C 180,E1 -11467.293,E2 -11467.293} C_VEL
LIN {X 0,Y 388.771,Z 354.295,A -85,B 0,C 180,E1 -11469.251,E2 -11469.251} C_VEL
LIN {X 0,Y 389.073,Z 351.515,A -85,B 0,C 180,E1 -11471.247,E2 -11471.247} C_VEL
LIN {X 0,Y 389.367,Z 348.051,A -85,B 0,C 180,E1 -11472.728,E2 -11472.728} C_VEL
LIN {X 0,Y 389.734,Z 343.366,A -85,B 0,C 180,E1 -11474.204,E2 -11474.204} C_VEL
LIN {X 0,Y 390.226,Z 337.314,A -85,B 0,C 180,E1 -11475.669,E2 -11475.669} C_VEL
LIN {X 0,Y 390.755,Z 330.835,A -85,B 0,C 180,E1 -11476.885,E2 -11476.885} C_VEL
LIN {X 0,Y 391.301,Z 324.024,A -85,B 0,C 180,E1 -11477.92,E2 -11477.92} C_VEL
LIN {X 0,Y 391.839,Z 316.323,A -85,B 0,C 180,E1 -11478.878,E2 -11478.878} C_VEL
LIN {X 0,Y 392.279,Z 309.412,A -85,B 0,C 180,E1 -11479.59,E2 -11479.59} C_VEL
LIN {X 0,Y 392.737,Z 300.852,A -85,B 0,C 180,E1 -11480.308,E2 -11480.308} C_VEL
LIN {X 0,Y 392.979,Z 293.295,A -85,B 0,C 180,E1 -11480.819,E2 -11480.819} C_VEL
LIN {X 0,Y 391.378,Z 283.828,A -85,B 0,C 180,E1 -11481.39,E2 -11481.39} C_VEL
LIN {X 0,Y 389.522,Z 275.453,A -85,B 0,C 180,E1 -11481.812,E2 -11481.812} C_VEL
LIN {X 0,Y 389.672,Z 268.296,A -85,B 0,C 180,E1 -11485.38,E2 -11485.38} C_VEL
LIN {X 0,Y 389.778,Z 262.029,A -85,B 0,C 180,E1 -11488.473,E2 -11488.473} C_VEL
LIN {X 0,Y 389.933,Z 254.913,A -85,B 0,C 180,E1 -11492.026,E2 -11492.026} C_VEL
LIN {X 0,Y 390.135,Z 246.332,A -85,B 0,C 180,E1 -11496.088,E2 -11496.088} C_VEL
LIN {X 0,Y 390.099,Z 240.412,A -85,B 0,C 180,E1 -11498.88,E2 -11498.88} C_VEL
LIN {X 0,Y 390.033,Z 239.905,A -85,B 0,C 180,E1 -11499.273,E2 -11499.273} C_VEL
LIN {X 0,Y 390.151,Z 239.889,A -85,B 0,C 180,E1 -11502.692,E2 -11502.692} C_VEL
LIN {X 0,Y 390.197,Z 239.882,A -85,B 0,C 180,E1 -11506.561,E2 -11506.561} C_VEL
LIN {X 0,Y 390.171,Z 239.887,A -85,B 0,C 180,E1 -11509.623,E2 -11509.623} C_VEL
LIN {X 0,Y 390.251,Z 239.876,A -85,B 0,C 180,E1 -11512.758,E2 -11512.758} C_VEL
LIN {X 0,Y 390.217,Z 239.879,A -85,B 0,C 180,E1 -11514.833,E2 -11514.833} C_VEL
LIN {X 0,Y 390.421,Z 239.855,A -85,B 0,C 180,E1 -11517.937,E2 -11517.937} C_VEL
LIN {X 0,Y 390.551,Z 239.837,A -85,B 0,C 180,E1 -11520,E2 -11520} C_VEL
LIN {X 0,Y 390.311,Z 239.867,A -85,B 0,C 180,E1 -11523.096,E2 -11523.096} C_VEL
LIN {X 0,Y 390.301,Z 239.868,A -85,B 0,C 180,E1 -11526.202,E2 -11526.202} C_VEL
LIN {X 0,Y 390.206,Z 239.88,A -85,B 0,C 180,E1 -11529.329,E2 -11529.329} C_VEL
LIN {X 0,Y 390.196,Z 239.88,A -85,B 0,C 180,E1 -11533.438,E2 -11533.438} C_VEL
LIN {X 0,Y 390.151,Z 239.887,A -85,B 0,C 180,E1 -11537.308,E2 -11537.308} C_VEL
LIN {X 0,Y 390.089,Z 239.895,A -85,B 0,C 180,E1 -11540.47,E2 -11540.47} C_VEL
LIN {X 0,Y 390.076,Z 239.895,A -85,B 0,C 180,E1 -11544.481,E2 -11544.481} C_VEL
LIN {X 0,Y 390.119,Z 239.891,A -85,B 0,C 180,E1 -11547.93,E2 -11547.93} C_VEL
LIN {X 0,Y 390.025,Z 239.901,A -85,B 0,C 180,E1 -11551.504,E2 -11551.504} C_VEL
LIN {X 0,Y 390.086,Z 239.893,A -85,B 0,C 180,E1 -11555.207,E2 -11555.207} C_VEL
LIN {X 0,Y 390.072,Z 239.896,A -85,B 0,C 180,E1 -11559.218,E2 -11559.218} C_VEL
LIN {X 0,Y 390.044,Z 239.899,A -85,B 0,C 180,E1 -11562.374,E2 -11562.374} C_VEL
LIN {X 0,Y 390.046,Z 239.903,A -85,B 0,C 180,E1 -11565.354,E2 -11565.354} C_VEL
LIN {X 0,Y 390.116,Z 240.054,A -85,B 0,C 180,E1 -11567.038,E2 -11567.038} C_VEL
LIN {X 0,Y 391.241,Z 246.513,A -85,B 0,C 180,E1 -11570.572,E2 -11570.572} C_VEL
LIN {X 0,Y 392.022,Z 251.331,A -85,B 0,C 180,E1 -11573.089,E2 -11573.089} C_VEL
LIN {X 0,Y 391.916,Z 256.369,A -85,B 0,C 180,E1 -11575.578,E2 -11575.578} C_VEL
LIN {X 0,Y 391.208,Z 262.74,A -85,B 0,C 180,E1 -11578.602,E2 -11578.602} C_VEL
LIN {X 0,Y 390.612,Z 269.703,A -85,B 0,C 180,E1 -11581.839,E2 -11581.839} C_VEL
LIN {X 0,Y 390.028,Z 277.815,A -85,B 0,C 180,E1 -11585.516,E2 -11585.516} C_VEL
LIN {X 0,Y 389.509,Z 286.472,A -85,B 0,C 180,E1 -11589.368,E2 -11589.368} C_VEL
LIN {X 0,Y 389.197,Z 292.991,A -85,B 0,C 180,E1 -11592.169,E2 -11592.169} C_VEL
LIN {X 0,Y 390.977,Z 307.069,A -85,B 0,C 180,E1 -11592.76,E2 -11592.76} C_VEL
LIN {X 0,Y 392.554,Z 320.617,A -85,B 0,C 180,E1 -11593.555,E2 -11593.555} C_VEL
LIN {X 0,Y 392.825,Z 325.623,A -85,B 0,C 180,E1 -11593.9,E2 -11593.9} C_VEL
LIN {X 0,Y 392.01,Z 337.082,A -85,B 0,C 180,E1 -11594.8,E2 -11594.8} C_VEL
LIN {X 0,Y 391.245,Z 347.771,A -85,B 0,C 180,E1 -11595.85,E2 -11595.85} C_VEL
LIN {X 0,Y 390.636,Z 357.336,A -85,B 0,C 180,E1 -11597.004,E2 -11597.004} C_VEL
LIN {X 0,Y 390.001,Z 366.239,A -85,B 0,C 180,E1 -11598.303,E2 -11598.303} C_VEL
LIN {X 0,Y 389.411,Z 374.979,A -85,B 0,C 180,E1 -11599.865,E2 -11599.865} C_VEL
LIN {X 0,Y 389.111,Z 381.969,A -85,B 0,C 180,E1 -11601.431,E2 -11601.431} C_VEL
LIN {X 0,Y 388.897,Z 388.368,A -85,B 0,C 180,E1 -11603.254,E2 -11603.254} C_VEL
LIN {X 0,Y 388.831,Z 392.528,A -85,B 0,C 180,E1 -11604.815,E2 -11604.815} C_VEL
LIN {X 0,Y 388.748,Z 394.681,A -85,B 0,C 180,E1 -11605.853,E2 -11605.853} C_VEL
LIN {X 0,Y 388.805,Z 396.354,A -85,B 0,C 180,E1 -11606.892,E2 -11606.892} C_VEL
LIN {X 0,Y 388.851,Z 397.601,A -85,B 0,C 180,E1 -11607.929,E2 -11607.929} C_VEL
LIN {X 0,Y 388.811,Z 398.421,A -85,B 0,C 180,E1 -11608.964,E2 -11608.964} C_VEL
LIN {X 0,Y 388.802,Z 398.778,A -85,B 0,C 180,E1 -11610,E2 -11610} C_VEL
LIN {X 0,Y 388.791,Z 398.715,A -85,B 0,C 180,E1 -11611.036,E2 -11611.036} C_VEL
LIN {X 0,Y 388.833,Z 398.247,A -85,B 0,C 180,E1 -11612.072,E2 -11612.072} C_VEL
LIN {X 0,Y 388.72,Z 397.353,A -85,B 0,C 180,E1 -11613.109,E2 -11613.109} C_VEL
LIN {X 0,Y 388.73,Z 396.002,A -85,B 0,C 180,E1 -11614.147,E2 -11614.147} C_VEL
LIN {X 0,Y 388.732,Z 393.055,A -85,B 0,C 180,E1 -11615.762,E2 -11615.762} C_VEL
LIN {X 0,Y 388.93,Z 389.324,A -85,B 0,C 180,E1 -11617.267,E2 -11617.267} C_VEL
LIN {X 0,Y 389.161,Z 384.344,A -85,B 0,C 180,E1 -11618.83,E2 -11618.83} C_VEL
LIN {X 0,Y 389.699,Z 376.965,A -85,B 0,C 180,E1 -11620.653,E2 -11620.653} C_VEL
LIN {X 0,Y 390.538,Z 369.077,A -85,B 0,C 180,E1 -11622.208,E2 -11622.208} C_VEL
LIN {X 0,Y 391.348,Z 359.354,A -85,B 0,C 180,E1 -11623.767,E2 -11623.767} C_VEL
LIN {X 0,Y 392.505,Z 348.479,A -85,B 0,C 180,E1 -11625.181,E2 -11625.181} C_VEL
LIN {X 0,Y 393.884,Z 336.184,A -85,B 0,C 180,E1 -11626.455,E2 -11626.455} C_VEL
LIN {X 0,Y 394.802,Z 325.683,A -85,B 0,C 180,E1 -11627.348,E2 -11627.348} C_VEL
LIN {X 0,Y 394.155,Z 312.561,A -85,B 0,C 180,E1 -11628.348,E2 -11628.348} C_VEL
LIN {X 0,Y 392.115,Z 299.681,A -85,B 0,C 180,E1 -11629.229,E2 -11629.229} C_VEL
LIN {X 0,Y 389.461,Z 288.389,A -85,B 0,C 180,E1 -11629.949,E2 -11629.949} C_VEL
LIN {X 0,Y 389.903,Z 280.969,A -85,B 0,C 180,E1 -11633.363,E2 -11633.363} C_VEL
LIN {X 0,Y 390.511,Z 274.072,A -85,B 0,C 180,E1 -11636.739,E2 -11636.739} C_VEL
LIN {X 0,Y 391.332,Z 267.141,A -85,B 0,C 180,E1 -11640.453,E2 -11640.453} C_VEL
LIN {X 0,Y 392.239,Z 261.665,A -85,B 0,C 180,E1 -11643.742,E2 -11643.742} C_VEL
LIN {X 0,Y 392.751,Z 257.887,A -85,B 0,C 180,E1 -11646.366,E2 -11646.366} C_VEL
LIN {X 0,Y 392.638,Z 255,A -85,B 0,C 180,E1 -11648.791,E2 -11648.791} C_VEL
LIN {X 0,Y 392.258,Z 252.411,A -85,B 0,C 180,E1 -11651.523,E2 -11651.523} C_VEL
LIN {X 0,Y 391.913,Z 250.378,A -85,B 0,C 180,E1 -11654.377,E2 -11654.377} C_VEL
LIN {X 0,Y 391.647,Z 248.955,A -85,B 0,C 180,E1 -11657.37,E2 -11657.37} C_VEL
LIN {X 0,Y 391.457,Z 248.211,A -85,B 0,C 180,E1 -11660.534,E2 -11660.534} C_VEL
LIN {X 0,Y 391.329,Z 248.139,A -85,B 0,C 180,E1 -11663.654,E2 -11663.654} C_VEL
LIN {X 0,Y 391.162,Z 248.513,A -85,B 0,C 180,E1 -11666.153,E2 -11666.153} C_VEL
LIN {X 0,Y 390.7,Z 249.649,A -85,B 0,C 180,E1 -11669.757,E2 -11669.757} C_VEL
LIN {X 0,Y 390.327,Z 251.237,A -85,B 0,C 180,E1 -11673.248,E2 -11673.248} C_VEL
LIN {X 0,Y 390.029,Z 253.157,A -85,B 0,C 180,E1 -11676.645,E2 -11676.645} C_VEL
LIN {X 0,Y 389.829,Z 255.306,A -85,B 0,C 180,E1 -11679.968,E2 -11679.968} C_VEL
LIN {X 0,Y 389.779,Z 256.189,A -85,B 0,C 180,E1 -11681.23,E2 -11681.23} C_VEL
LIN {X 0,Y 390.847,Z 259.206,A -85,B 0,C 180,E1 -11681.469,E2 -11681.469} C_VEL
LIN {X 0,Y 395.191,Z 271.225,A -85,B 0,C 180,E1 -11682.48,E2 -11682.48} C_VEL
LIN {X 0,Y 397.098,Z 279.323,A -85,B 0,C 180,E1 -11683.174,E2 -11683.174} C_VEL
LIN {X 0,Y 396.124,Z 291.486,A -85,B 0,C 180,E1 -11684.102,E2 -11684.102} C_VEL
LIN {X 0,Y 394.844,Z 303.915,A -85,B 0,C 180,E1 -11685.307,E2 -11685.307} C_VEL
LIN {X 0,Y 393.683,Z 314.43,A -85,B 0,C 180,E1 -11686.581,E2 -11686.581} C_VEL
LIN {X 0,Y 392.546,Z 324.565,A -85,B 0,C 180,E1 -11688.118,E2 -11688.118} C_VEL
LIN {X 0,Y 391.495,Z 332.799,A -85,B 0,C 180,E1 -11689.658,E2 -11689.658} C_VEL
LIN {X 0,Y 390.801,Z 339.397,A -85,B 0,C 180,E1 -11691.207,E2 -11691.207} C_VEL
LIN {X 0,Y 390.005,Z 344.728,A -85,B 0,C 180,E1 -11692.753,E2 -11692.753} C_VEL
LIN {X 0,Y 389.793,Z 348.854,A -85,B 0,C 180,E1 -11694.309,E2 -11694.309} C_VEL
LIN {X 0,Y 389.508,Z 351.964,A -85,B 0,C 180,E1 -11695.861,E2 -11695.861} C_VEL
LIN {X 0,Y 389.377,Z 353.486,A -85,B 0,C 180,E1 -11696.896,E2 -11696.896} C_VEL
LIN {X 0,Y 389.086,Z 354.621,A -85,B 0,C 180,E1 -11697.93,E2 -11697.93} C_VEL
LIN {X 0,Y 388.93,Z 355.304,A -85,B 0,C 180,E1 -11698.965,E2 -11698.965} C_VEL
LIN {X 0,Y 388.832,Z 355.449,A -85,B 0,C 180,E1 -11701.036,E2 -11701.036} C_VEL
LIN {X 0,Y 388.892,Z 354.92,A -85,B 0,C 180,E1 -11702.071,E2 -11702.071} C_VEL
LIN {X 0,Y 388.945,Z 353.942,A -85,B 0,C 180,E1 -11703.108,E2 -11703.108} C_VEL
LIN {X 0,Y 388.902,Z 352.559,A -85,B 0,C 180,E1 -11704.145,E2 -11704.145} C_VEL
LIN {X 0,Y 389.074,Z 349.664,A -85,B 0,C 180,E1 -11705.702,E2 -11705.702} C_VEL
LIN {X 0,Y 389.233,Z 345.719,A -85,B 0,C 180,E1 -11707.261,E2 -11707.261} C_VEL
LIN {X 0,Y 389.527,Z 340.613,A -85,B 0,C 180,E1 -11708.822,E2 -11708.822} C_VEL
LIN {X 0,Y 389.93,Z 334.204,A -85,B 0,C 180,E1 -11710.384,E2 -11710.384} C_VEL
LIN {X 0,Y 390.475,Z 326.212,A -85,B 0,C 180,E1 -11711.946,E2 -11711.946} C_VEL
LIN {X 0,Y 391.056,Z 318.086,A -85,B 0,C 180,E1 -11713.247,E2 -11713.247} C_VEL
LIN {X 0,Y 391.649,Z 308.241,A -85,B 0,C 180,E1 -11714.55,E2 -11714.55} C_VEL
LIN {X 0,Y 392.388,Z 297.382,A -85,B 0,C 180,E1 -11715.718,E2 -11715.718} C_VEL
LIN {X 0,Y 393.24,Z 285.288,A -85,B 0,C 180,E1 -11716.75,E2 -11716.75} C_VEL
LIN {X 0,Y 393.716,Z 274.472,A -85,B 0,C 180,E1 -11717.488,E2 -11717.488} C_VEL
LIN {X 0,Y 391.105,Z 261.37,A -85,B 0,C 180,E1 -11718.272,E2 -11718.272} C_VEL
LIN {X 0,Y 388.977,Z 251.165,A -85,B 0,C 180,E1 -11718.774,E2 -11718.774} C_VEL
LIN {X 0,Y 388.989,Z 247.463,A -85,B 0,C 180,E1 -11722.298,E2 -11722.298} C_VEL
LIN {X 0,Y 389.153,Z 243.967,A -85,B 0,C 180,E1 -11725.686,E2 -11725.686} C_VEL
LIN {X 0,Y 389.173,Z 240.468,A -85,B 0,C 180,E1 -11729.182,E2 -11729.182} C_VEL
LIN {X 0,Y 389.25,Z 239.999,A -85,B 0,C 180,E1 -11730.368,E2 -11730.368} C_VEL
LIN {X 0,Y 389.749,Z 239.936,A -85,B 0,C 180,E1 -11733.954,E2 -11733.954} C_VEL
LIN {X 0,Y 389.965,Z 239.908,A -85,B 0,C 180,E1 -11736.494,E2 -11736.494} C_VEL
LIN {X 0,Y 390.063,Z 239.898,A -85,B 0,C 180,E1 -11739.216,E2 -11739.216} C_VEL
LIN {X 0,Y 390.043,Z 239.898,A -85,B 0,C 180,E1 -11742.373,E2 -11742.373} C_VEL
LIN {X 0,Y 390.047,Z 239.9,A -85,B 0,C 180,E1 -11745.354,E2 -11745.354} C_VEL
LIN {X 0,Y 390.02,Z 239.901,A -85,B 0,C 180,E1 -11748.185,E2 -11748.185} C_VEL
LIN {X 0,Y 390.059,Z 239.901,A -85,B 0,C 180,E1 -11750.903,E2 -11750.903} C_VEL
LIN {X 0,Y 390.071,Z 239.899,A -85,B 0,C 180,E1 -11754.791,E2 -11754.791} C_VEL
LIN {X 0,Y 390.026,Z 239.904,A -85,B 0,C 180,E1 -11758.496,E2 -11758.496} C_VEL
LIN {X 0,Y 390.078,Z 239.895,A -85,B 0,C 180,E1 -11762.067,E2 -11762.067} C_VEL
